Fanuc TP program (LS listing): test_parallel.ls

/PROG  test_parallel
/ATTR
COMMENT	= "18-08-08 11:10:22";
PROG_SIZE	= 0;
DEFAULT_GROUP	= 1, 1, *, *, *;
/APPL
    ARC Welding Equipment: 1, *, *, *, *;
/MN
   1:  CALL HOME_ALL;
   1:  UFRAME_NUM = 1;
   1:  UTOOL_NUM = 3;
   1:  COL GUARD ADJUST 150;
   1:  PR[91] = PR[90];
   1:  PR[GP1:91,1] = PR[GP1:90,1] + 65.993;
   1:  PR[GP1:91,2] = PR[GP1:90,2] + 95.281;
   1:  PR[GP1:91,3] = PR[GP1:90,3] + 0.900;
   1:L PR[91] 10mm/sec FINE;
   1:  PR[GP1:91,1] = PR[GP1:90,1] + 66.256;
   1:  PR[GP1:91,2] = PR[GP1:90,2] + 95.138;
   1:L PR[91] 10mm/sec FINE;
   1:  PR[GP1:91,1] = PR[GP1:90,1] + 70.899;
   1:  PR[GP1:91,2] = PR[GP1:90,2] + 93.080;
   1:L PR[91] 10mm/sec FINE;
   1:  PR[GP1:91,1] = PR[GP1:90,1] + 71.182;
   1:  PR[GP1:91,2] = PR[GP1:90,2] + 92.981;
   1:L PR[91] 10mm/sec FINE;
   1:  PR[GP1:91,1] = PR[GP1:90,1] + 71.477;
   1:  PR[GP1:91,2] = PR[GP1:90,2] + 92.931;
   1:L PR[91] 10mm/sec FINE;
   1:  PR[GP1:91,1] = PR[GP1:90,1] + 76.535;
   1:  PR[GP1:91,2] = PR[GP1:90,2] + 92.486;
   1:L PR[91] 10mm/sec FINE;
   1:  PR[GP1:91,1] = PR[GP1:90,1] + 76.835;
   1:  PR[GP1:91,2] = PR[GP1:90,2] + 92.484;
   1:L PR[91] 10mm/sec FINE;
   1:  PR[GP1:91,1] = PR[GP1:90,1] + 77.130;
   1:  PR[GP1:91,2] = PR[GP1:90,2] + 92.532;
   1:L PR[91] 10mm/sec FINE;
   1:  PR[GP1:91,1] = PR[GP1:90,1] + 82.061;
   1:  PR[GP1:91,2] = PR[GP1:90,2] + 93.748;
   1:L PR[91] 10mm/sec FINE;
   1:  PR[GP1:91,1] = PR[GP1:90,1] + 82.344;
   1:  PR[GP1:91,2] = PR[GP1:90,2] + 93.843;
   1:L PR[91] 10mm/sec FINE;
   1:  PR[GP1:91,1] = PR[GP1:90,1] + 82.609;
   1:  PR[GP1:91,2] = PR[GP1:90,2] + 93.984;
   1:L PR[91] 10mm/sec FINE;
   1:  PR[GP1:91,1] = PR[GP1:90,1] + 86.880;
   1:  PR[GP1:91,2] = PR[GP1:90,2] + 96.730;
   1:L PR[91] 10mm/sec FINE;
   1:  PR[GP1:91,1] = PR[GP1:90,1] + 87.118;
   1:  PR[GP1:91,2] = PR[GP1:90,2] + 96.912;
   1:L PR[91] 10mm/sec FINE;
   1:  PR[GP1:91,1] = PR[GP1:90,1] + 87.322;
   1:  PR[GP1:91,2] = PR[GP1:90,2] + 97.130;
   1:L PR[91] 10mm/sec FINE;
   1:  PR[GP1:91,1] = PR[GP1:90,1] + 90.476;
   1:  PR[GP1:91,2] = PR[GP1:90,2] + 101.111;
   1:L PR[91] 10mm/sec FINE;
   1:  PR[GP1:91,1] = PR[GP1:90,1] + 90.641;
   1:  PR[GP1:91,2] = PR[GP1:90,2] + 101.360;
   1:L PR[91] 10mm/sec FINE;
   1:  PR[GP1:91,1] = PR[GP1:90,1] + 90.764;
   1:  PR[GP1:91,2] = PR[GP1:90,2] + 101.633;
   1:L PR[91] 10mm/sec FINE;
   1:  PR[GP1:91,1] = PR[GP1:90,1] + 92.459;
   1:  PR[GP1:91,2] = PR[GP1:90,2] + 106.415;
   1:L PR[91] 10mm/sec FINE;
   1:  PR[GP1:91,1] = PR[GP1:90,1] + 92.544;
   1:  PR[GP1:91,2] = PR[GP1:90,2] + 106.735;
   1:L PR[91] 10mm/sec FINE;
   1:  PR[GP1:91,1] = PR[GP1:90,1] + 93.026;
   1:  PR[GP1:91,2] = PR[GP1:90,2] + 107.850;
   1:L PR[91] 10mm/sec FINE;
   1:  PR[GP1:91,1] = PR[GP1:90,1] + 93.981;
   1:  PR[GP1:91,2] = PR[GP1:90,2] + 108.650;
   1:L PR[91] 10mm/sec FINE;
   1:  PR[GP1:91,1] = PR[GP1:90,1] + 95.171;
   1:  PR[GP1:91,2] = PR[GP1:90,2] + 108.932;
   1:L PR[91] 10mm/sec FINE;
   1:  PR[GP1:91,1] = PR[GP1:90,1] + 95.835;
   1:L PR[91] 10mm/sec FINE;
   1:  PR[GP1:91,1] = PR[GP1:90,1] + 97.026;
   1:  PR[GP1:91,2] = PR[GP1:90,2] + 108.650;
   1:L PR[91] 10mm/sec FINE;
   1:  PR[GP1:91,1] = PR[GP1:90,1] + 97.981;
   1:  PR[GP1:91,2] = PR[GP1:90,2] + 107.850;
   1:L PR[91] 10mm/sec FINE;
   1:  PR[GP1:91,1] = PR[GP1:90,1] + 98.460;
   1:  PR[GP1:91,2] = PR[GP1:90,2] + 106.743;
   1:L PR[91] 10mm/sec FINE;
   1:  PR[GP1:91,1] = PR[GP1:90,1] + 100.166;
   1:  PR[GP1:91,2] = PR[GP1:90,2] + 101.928;
   1:L PR[91] 10mm/sec FINE;
   1:  PR[GP1:91,1] = PR[GP1:90,1] + 100.215;
   1:  PR[GP1:91,2] = PR[GP1:90,2] + 101.718;
   1:L PR[91] 10mm/sec FINE;
   1:  PR[GP1:91,1] = PR[GP1:90,1] + 100.280;
   1:  PR[GP1:91,2] = PR[GP1:90,2] + 101.535;
   1:L PR[91] 10mm/sec FINE;
   1:  PR[GP1:91,1] = PR[GP1:90,1] + 100.360;
   1:  PR[GP1:91,2] = PR[GP1:90,2] + 101.370;
   1:L PR[91] 10mm/sec FINE;
   1:  PR[GP1:91,1] = PR[GP1:90,1] + 103.517;
   1:  PR[GP1:91,2] = PR[GP1:90,2] + 97.385;
   1:L PR[91] 10mm/sec FINE;
   1:  PR[GP1:91,1] = PR[GP1:90,1] + 103.631;
   1:  PR[GP1:91,2] = PR[GP1:90,2] + 97.202;
   1:L PR[91] 10mm/sec FINE;
   1:  PR[GP1:91,1] = PR[GP1:90,1] + 103.752;
   1:  PR[GP1:91,2] = PR[GP1:90,2] + 97.049;
   1:L PR[91] 10mm/sec FINE;
   1:  PR[GP1:91,1] = PR[GP1:90,1] + 103.881;
   1:  PR[GP1:91,2] = PR[GP1:90,2] + 96.919;
   1:L PR[91] 10mm/sec FINE;
   1:  PR[GP1:91,1] = PR[GP1:90,1] + 108.157;
   1:  PR[GP1:91,2] = PR[GP1:90,2] + 94.170;
   1:L PR[91] 10mm/sec FINE;
   1:  PR[GP1:91,1] = PR[GP1:90,1] + 108.325;
   1:  PR[GP1:91,2] = PR[GP1:90,2] + 94.034;
   1:L PR[91] 10mm/sec FINE;
   1:  PR[GP1:91,1] = PR[GP1:90,1] + 108.488;
   1:  PR[GP1:91,2] = PR[GP1:90,2] + 93.929;
   1:L PR[91] 10mm/sec FINE;
   1:  PR[GP1:91,1] = PR[GP1:90,1] + 108.652;
   1:  PR[GP1:91,2] = PR[GP1:90,2] + 93.848;
   1:L PR[91] 10mm/sec FINE;
   1:  PR[GP1:91,1] = PR[GP1:90,1] + 113.587;
   1:  PR[GP1:91,2] = PR[GP1:90,2] + 92.631;
   1:L PR[91] 10mm/sec FINE;
   1:  PR[GP1:91,1] = PR[GP1:90,1] + 113.790;
   1:  PR[GP1:91,2] = PR[GP1:90,2] + 92.556;
   1:L PR[91] 10mm/sec FINE;
   1:  PR[GP1:91,1] = PR[GP1:90,1] + 113.978;
   1:  PR[GP1:91,2] = PR[GP1:90,2] + 92.510;
   1:L PR[91] 10mm/sec FINE;
   1:  PR[GP1:91,1] = PR[GP1:90,1] + 114.160;
   1:  PR[GP1:91,2] = PR[GP1:90,2] + 92.486;
   1:L PR[91] 10mm/sec FINE;
   1:  PR[GP1:91,1] = PR[GP1:90,1] + 119.224;
   1:  PR[GP1:91,2] = PR[GP1:90,2] + 92.931;
   1:L PR[91] 10mm/sec FINE;
   1:  PR[GP1:91,1] = PR[GP1:90,1] + 119.440;
   1:  PR[GP1:91,2] = PR[GP1:90,2] + 92.926;
   1:L PR[91] 10mm/sec FINE;
   1:  PR[GP1:91,1] = PR[GP1:90,1] + 119.633;
   1:  PR[GP1:91,2] = PR[GP1:90,2] + 92.943;
   1:L PR[91] 10mm/sec FINE;
   1:  PR[GP1:91,1] = PR[GP1:90,1] + 119.813;
   1:  PR[GP1:91,2] = PR[GP1:90,2] + 92.979;
   1:L PR[91] 10mm/sec FINE;
   1:  PR[GP1:91,1] = PR[GP1:90,1] + 124.460;
   1:  PR[GP1:91,2] = PR[GP1:90,2] + 95.038;
   1:L PR[91] 10mm/sec FINE;
   1:  PR[GP1:91,1] = PR[GP1:90,1] + 124.666;
   1:  PR[GP1:91,2] = PR[GP1:90,2] + 95.104;
   1:L PR[91] 10mm/sec FINE;
   1:  PR[GP1:91,1] = PR[GP1:90,1] + 124.844;
   1:  PR[GP1:91,2] = PR[GP1:90,2] + 95.182;
   1:L PR[91] 10mm/sec FINE;
   1:  PR[GP1:91,1] = PR[GP1:90,1] + 125.002;
   1:  PR[GP1:91,2] = PR[GP1:90,2] + 95.275;
   1:L PR[91] 10mm/sec FINE;
   1:  PR[GP1:91,1] = PR[GP1:90,1] + 128.734;
   1:  PR[GP1:91,2] = PR[GP1:90,2] + 98.728;
   1:L PR[91] 10mm/sec FINE;
   1:  PR[GP1:91,1] = PR[GP1:90,1] + 128.907;
   1:  PR[GP1:91,2] = PR[GP1:90,2] + 98.856;
   1:L PR[91] 10mm/sec FINE;
   1:  PR[GP1:91,1] = PR[GP1:90,1] + 129.050;
   1:  PR[GP1:91,2] = PR[GP1:90,2] + 98.988;
   1:L PR[91] 10mm/sec FINE;
   1:  PR[GP1:91,1] = PR[GP1:90,1] + 129.170;
   1:  PR[GP1:91,2] = PR[GP1:90,2] + 99.127;
   1:L PR[91] 10mm/sec FINE;
   1:  PR[GP1:91,1] = PR[GP1:90,1] + 131.584;
   1:  PR[GP1:91,2] = PR[GP1:90,2] + 103.603;
   1:L PR[91] 10mm/sec FINE;
   1:  PR[GP1:91,1] = PR[GP1:90,1] + 131.706;
   1:  PR[GP1:91,2] = PR[GP1:90,2] + 103.781;
   1:L PR[91] 10mm/sec FINE;
   1:  PR[GP1:91,1] = PR[GP1:90,1] + 131.798;
   1:  PR[GP1:91,2] = PR[GP1:90,2] + 103.951;
   1:L PR[91] 10mm/sec FINE;
   1:  PR[GP1:91,1] = PR[GP1:90,1] + 131.867;
   1:  PR[GP1:91,2] = PR[GP1:90,2] + 104.121;
   1:L PR[91] 10mm/sec FINE;
   1:  PR[GP1:91,1] = PR[GP1:90,1] + 132.702;
   1:  PR[GP1:91,2] = PR[GP1:90,2] + 109.139;
   1:L PR[91] 10mm/sec FINE;
   1:  PR[GP1:91,1] = PR[GP1:90,1] + 132.760;
   1:  PR[GP1:91,2] = PR[GP1:90,2] + 109.347;
   1:L PR[91] 10mm/sec FINE;
   1:  PR[GP1:91,1] = PR[GP1:90,1] + 132.792;
   1:  PR[GP1:91,2] = PR[GP1:90,2] + 109.538;
   1:L PR[91] 10mm/sec FINE;
   1:  PR[GP1:91,1] = PR[GP1:90,1] + 132.802;
   1:  PR[GP1:91,2] = PR[GP1:90,2] + 109.721;
   1:L PR[91] 10mm/sec FINE;
   1:  PR[GP1:91,1] = PR[GP1:90,1] + 131.968;
   1:  PR[GP1:91,2] = PR[GP1:90,2] + 114.734;
   1:L PR[91] 10mm/sec FINE;
   1:  PR[GP1:91,1] = PR[GP1:90,1] + 131.931;
   1:  PR[GP1:91,2] = PR[GP1:90,2] + 115.108;
   1:L PR[91] 10mm/sec FINE;
   1:  PR[GP1:91,1] = PR[GP1:90,1] + 131.829;
   1:  PR[GP1:91,2] = PR[GP1:90,2] + 115.442;
   1:L PR[91] 10mm/sec FINE;
   1:  PR[GP1:91,1] = PR[GP1:90,1] + 129.241;
   1:  PR[GP1:91,2] = PR[GP1:90,2] + 120.241;
   1:L PR[91] 10mm/sec FINE;
   1:  PR[GP1:91,1] = PR[GP1:90,1] + 129.179;
   1:  PR[GP1:91,2] = PR[GP1:90,2] + 120.327;
   1:L PR[91] 10mm/sec FINE;
   1:  PR[GP1:91,1] = PR[GP1:90,1] + 129.019;
   1:  PR[GP1:91,2] = PR[GP1:90,2] + 120.507;
   1:L PR[91] 10mm/sec FINE;
   1:  PR[GP1:91,1] = PR[GP1:90,1] + 125.292;
   1:  PR[GP1:91,2] = PR[GP1:90,2] + 123.956;
   1:L PR[91] 10mm/sec FINE;
   1:  PR[GP1:91,1] = PR[GP1:90,1] + 125.015;
   1:  PR[GP1:91,2] = PR[GP1:90,2] + 124.180;
   1:L PR[91] 10mm/sec FINE;
   1:  PR[GP1:91,1] = PR[GP1:90,1] + 120.376;
   1:  PR[GP1:91,2] = PR[GP1:90,2] + 126.236;
   1:L PR[91] 10mm/sec FINE;
   1:  PR[GP1:91,1] = PR[GP1:90,1] + 120.040;
   1:  PR[GP1:91,2] = PR[GP1:90,2] + 126.412;
   1:L PR[91] 10mm/sec FINE;
   1:  PR[GP1:91,1] = PR[GP1:90,1] + 119.820;
   1:  PR[GP1:91,2] = PR[GP1:90,2] + 126.484;
   1:L PR[91] 10mm/sec FINE;
   1:  PR[GP1:91,1] = PR[GP1:90,1] + 119.714;
   1:  PR[GP1:91,2] = PR[GP1:90,2] + 126.508;
   1:L PR[91] 10mm/sec FINE;
   1:  PR[GP1:91,1] = PR[GP1:90,1] + 114.278;
   1:  PR[GP1:91,2] = PR[GP1:90,2] + 126.985;
   1:L PR[91] 10mm/sec FINE;
   1:  PR[GP1:91,1] = PR[GP1:90,1] + 114.174;
   1:  PR[GP1:91,2] = PR[GP1:90,2] + 126.981;
   1:L PR[91] 10mm/sec FINE;
   1:  PR[GP1:91,1] = PR[GP1:90,1] + 113.934;
   1:  PR[GP1:91,2] = PR[GP1:90,2] + 126.946;
   1:L PR[91] 10mm/sec FINE;
   1:  PR[GP1:91,1] = PR[GP1:90,1] + 109.004;
   1:  PR[GP1:91,2] = PR[GP1:90,2] + 125.730;
   1:L PR[91] 10mm/sec FINE;
   1:  PR[GP1:91,1] = PR[GP1:90,1] + 108.669;
   1:  PR[GP1:91,2] = PR[GP1:90,2] + 125.623;
   1:L PR[91] 10mm/sec FINE;
   1:  PR[GP1:91,1] = PR[GP1:90,1] + 104.397;
   1:  PR[GP1:91,2] = PR[GP1:90,2] + 122.877;
   1:L PR[91] 10mm/sec FINE;
   1:  PR[GP1:91,1] = PR[GP1:90,1] + 104.066;
   1:  PR[GP1:91,2] = PR[GP1:90,2] + 122.693;
   1:L PR[91] 10mm/sec FINE;
   1:  PR[GP1:91,1] = PR[GP1:90,1] + 103.886;
   1:  PR[GP1:91,2] = PR[GP1:90,2] + 122.551;
   1:L PR[91] 10mm/sec FINE;
   1:  PR[GP1:91,1] = PR[GP1:90,1] + 103.806;
   1:  PR[GP1:91,2] = PR[GP1:90,2] + 122.474;
   1:L PR[91] 10mm/sec FINE;
   1:  PR[GP1:91,1] = PR[GP1:90,1] + 100.418;
   1:  PR[GP1:91,2] = PR[GP1:90,2] + 118.195;
   1:L PR[91] 10mm/sec FINE;
   1:  PR[GP1:91,1] = PR[GP1:90,1] + 100.366;
   1:  PR[GP1:91,2] = PR[GP1:90,2] + 118.108;
   1:L PR[91] 10mm/sec FINE;
   1:  PR[GP1:91,1] = PR[GP1:90,1] + 100.262;
   1:  PR[GP1:91,2] = PR[GP1:90,2] + 117.886;
   1:L PR[91] 10mm/sec FINE;
   1:  PR[GP1:91,1] = PR[GP1:90,1] + 98.568;
   1:  PR[GP1:91,2] = PR[GP1:90,2] + 113.104;
   1:L PR[91] 10mm/sec FINE;
   1:  PR[GP1:91,1] = PR[GP1:90,1] + 98.462;
   1:  PR[GP1:91,2] = PR[GP1:90,2] + 112.728;
   1:L PR[91] 10mm/sec FINE;
   1:  PR[GP1:91,1] = PR[GP1:90,1] + 97.981;
   1:  PR[GP1:91,2] = PR[GP1:90,2] + 111.615;
   1:L PR[91] 10mm/sec FINE;
   1:  PR[GP1:91,1] = PR[GP1:90,1] + 97.026;
   1:  PR[GP1:91,2] = PR[GP1:90,2] + 110.814;
   1:L PR[91] 10mm/sec FINE;
   1:  PR[GP1:91,1] = PR[GP1:90,1] + 95.835;
   1:  PR[GP1:91,2] = PR[GP1:90,2] + 110.532;
   1:L PR[91] 10mm/sec FINE;
   1:  PR[GP1:91,1] = PR[GP1:90,1] + 95.171;
   1:L PR[91] 10mm/sec FINE;
   1:  PR[GP1:91,1] = PR[GP1:90,1] + 93.981;
   1:  PR[GP1:91,2] = PR[GP1:90,2] + 110.814;
   1:L PR[91] 10mm/sec FINE;
   1:  PR[GP1:91,1] = PR[GP1:90,1] + 93.026;
   1:  PR[GP1:91,2] = PR[GP1:90,2] + 111.615;
   1:L PR[91] 10mm/sec FINE;
   1:  PR[GP1:91,1] = PR[GP1:90,1] + 92.547;
   1:  PR[GP1:91,2] = PR[GP1:90,2] + 112.721;
   1:L PR[91] 10mm/sec FINE;
   1:  PR[GP1:91,1] = PR[GP1:90,1] + 90.842;
   1:  PR[GP1:91,2] = PR[GP1:90,2] + 117.534;
   1:L PR[91] 10mm/sec FINE;
   1:  PR[GP1:91,1] = PR[GP1:90,1] + 90.761;
   1:  PR[GP1:91,2] = PR[GP1:90,2] + 117.840;
   1:L PR[91] 10mm/sec FINE;
   1:  PR[GP1:91,1] = PR[GP1:90,1] + 90.645;
   1:  PR[GP1:91,2] = PR[GP1:90,2] + 118.097;
   1:L PR[91] 10mm/sec FINE;
   1:  PR[GP1:91,1] = PR[GP1:90,1] + 87.492;
   1:  PR[GP1:91,2] = PR[GP1:90,2] + 122.078;
   1:L PR[91] 10mm/sec FINE;
   1:  PR[GP1:91,1] = PR[GP1:90,1] + 87.317;
   1:  PR[GP1:91,2] = PR[GP1:90,2] + 122.340;
   1:L PR[91] 10mm/sec FINE;
   1:  PR[GP1:91,1] = PR[GP1:90,1] + 87.123;
   1:  PR[GP1:91,2] = PR[GP1:90,2] + 122.547;
   1:L PR[91] 10mm/sec FINE;
   1:  PR[GP1:91,1] = PR[GP1:90,1] + 82.852;
   1:  PR[GP1:91,2] = PR[GP1:90,2] + 125.293;
   1:L PR[91] 10mm/sec FINE;
   1:  PR[GP1:91,1] = PR[GP1:90,1] + 82.601;
   1:  PR[GP1:91,2] = PR[GP1:90,2] + 125.485;
   1:L PR[91] 10mm/sec FINE;
   1:  PR[GP1:91,1] = PR[GP1:90,1] + 82.352;
   1:  PR[GP1:91,2] = PR[GP1:90,2] + 125.617;
   1:L PR[91] 10mm/sec FINE;
   1:  PR[GP1:91,1] = PR[GP1:90,1] + 77.421;
   1:  PR[GP1:91,2] = PR[GP1:90,2] + 126.834;
   1:L PR[91] 10mm/sec FINE;
   1:  PR[GP1:91,1] = PR[GP1:90,1] + 77.122;
   1:  PR[GP1:91,2] = PR[GP1:90,2] + 126.934;
   1:L PR[91] 10mm/sec FINE;
   1:  PR[GP1:91,1] = PR[GP1:90,1] + 76.843;
   1:  PR[GP1:91,2] = PR[GP1:90,2] + 126.979;
   1:L PR[91] 10mm/sec FINE;
   1:  PR[GP1:91,1] = PR[GP1:90,1] + 71.784;
   1:  PR[GP1:91,2] = PR[GP1:90,2] + 126.534;
   1:L PR[91] 10mm/sec FINE;
   1:  PR[GP1:91,1] = PR[GP1:90,1] + 71.468;
   1:  PR[GP1:91,2] = PR[GP1:90,2] + 126.532;
   1:L PR[91] 10mm/sec FINE;
   1:  PR[GP1:91,1] = PR[GP1:90,1] + 71.190;
   1:  PR[GP1:91,2] = PR[GP1:90,2] + 126.484;
   1:L PR[91] 10mm/sec FINE;
   1:  PR[GP1:91,1] = PR[GP1:90,1] + 66.547;
   1:  PR[GP1:91,2] = PR[GP1:90,2] + 124.426;
   1:L PR[91] 10mm/sec FINE;
   1:  PR[GP1:91,1] = PR[GP1:90,1] + 66.249;
   1:  PR[GP1:91,2] = PR[GP1:90,2] + 124.323;
   1:L PR[91] 10mm/sec FINE;
   1:  PR[GP1:91,1] = PR[GP1:90,1] + 66.001;
   1:  PR[GP1:91,2] = PR[GP1:90,2] + 124.187;
   1:L PR[91] 10mm/sec FINE;
   1:  PR[GP1:91,1] = PR[GP1:90,1] + 62.274;
   1:  PR[GP1:91,2] = PR[GP1:90,2] + 120.737;
   1:L PR[91] 10mm/sec FINE;
   1:  PR[GP1:91,1] = PR[GP1:90,1] + 62.025;
   1:  PR[GP1:91,2] = PR[GP1:90,2] + 120.542;
   1:L PR[91] 10mm/sec FINE;
   1:  PR[GP1:91,1] = PR[GP1:90,1] + 61.834;
   1:  PR[GP1:91,2] = PR[GP1:90,2] + 120.334;
   1:L PR[91] 10mm/sec FINE;
   1:  PR[GP1:91,1] = PR[GP1:90,1] + 59.424;
   1:  PR[GP1:91,2] = PR[GP1:90,2] + 115.863;
   1:L PR[91] 10mm/sec FINE;
   1:  PR[GP1:91,1] = PR[GP1:90,1] + 59.252;
   1:  PR[GP1:91,2] = PR[GP1:90,2] + 115.598;
   1:L PR[91] 10mm/sec FINE;
   1:  PR[GP1:91,1] = PR[GP1:90,1] + 59.139;
   1:  PR[GP1:91,2] = PR[GP1:90,2] + 115.339;
   1:L PR[91] 10mm/sec FINE;
   1:  PR[GP1:91,1] = PR[GP1:90,1] + 58.305;
   1:  PR[GP1:91,2] = PR[GP1:90,2] + 110.328;
   1:L PR[91] 10mm/sec FINE;
   1:  PR[GP1:91,1] = PR[GP1:90,1] + 58.228;
   1:  PR[GP1:91,2] = PR[GP1:90,2] + 110.022;
   1:L PR[91] 10mm/sec FINE;
   1:  PR[GP1:91,1] = PR[GP1:90,1] + 58.205;
   1:  PR[GP1:91,2] = PR[GP1:90,2] + 109.741;
   1:L PR[91] 10mm/sec FINE;
   1:  PR[GP1:91,1] = PR[GP1:90,1] + 59.038;
   1:  PR[GP1:91,2] = PR[GP1:90,2] + 104.730;
   1:L PR[91] 10mm/sec FINE;
   1:  PR[GP1:91,1] = PR[GP1:90,1] + 59.064;
   1:  PR[GP1:91,2] = PR[GP1:90,2] + 104.415;
   1:L PR[91] 10mm/sec FINE;
   1:  PR[GP1:91,1] = PR[GP1:90,1] + 59.135;
   1:  PR[GP1:91,2] = PR[GP1:90,2] + 104.133;
   1:L PR[91] 10mm/sec FINE;
   1:  PR[GP1:91,1] = PR[GP1:90,1] + 59.255;
   1:  PR[GP1:91,2] = PR[GP1:90,2] + 103.859;
   1:L PR[91] 10mm/sec FINE;
   1:  PR[GP1:91,1] = PR[GP1:90,1] + 61.665;
   1:  PR[GP1:91,2] = PR[GP1:90,2] + 99.388;
   1:L PR[91] 10mm/sec FINE;
   1:  PR[GP1:91,1] = PR[GP1:90,1] + 61.829;
   1:  PR[GP1:91,2] = PR[GP1:90,2] + 99.137;
   1:L PR[91] 10mm/sec FINE;
   1:  PR[GP1:91,1] = PR[GP1:90,1] + 62.031;
   1:  PR[GP1:91,2] = PR[GP1:90,2] + 98.916;
   1:L PR[91] 10mm/sec FINE;
   1:  PR[GP1:91,1] = PR[GP1:90,1] + 65.758;
   1:  PR[GP1:91,2] = PR[GP1:90,2] + 95.466;
   1:L PR[91] 10mm/sec FINE;
   1:  PR[GP1:91,1] = PR[GP1:90,1] + 65.993;
   1:  PR[GP1:91,2] = PR[GP1:90,2] + 95.281;
   1:L PR[91] 10mm/sec FINE;
   1:  PR[GP1:91,1] = PR[GP1:90,1] + 66.856;
   1:  PR[GP1:91,2] = PR[GP1:90,2] + 94.811;
   1:  PR[GP1:91,3] = PR[GP1:90,3] + 1.900;
   1:L PR[91] 10mm/sec FINE;
   1:  PR[GP1:91,1] = PR[GP1:90,1] + 70.252;
   1:  PR[GP1:91,2] = PR[GP1:90,2] + 93.305;
   1:L PR[91] 10mm/sec FINE;
   1:  PR[GP1:91,1] = PR[GP1:90,1] + 71.181;
   1:  PR[GP1:91,2] = PR[GP1:90,2] + 92.982;
   1:L PR[91] 10mm/sec FINE;
   1:  PR[GP1:91,1] = PR[GP1:90,1] + 72.150;
   1:  PR[GP1:91,2] = PR[GP1:90,2] + 92.815;
   1:L PR[91] 10mm/sec FINE;
   1:  PR[GP1:91,1] = PR[GP1:90,1] + 75.850;
   1:  PR[GP1:91,2] = PR[GP1:90,2] + 92.490;
   1:L PR[91] 10mm/sec FINE;
   1:  PR[GP1:91,1] = PR[GP1:90,1] + 76.834;
   1:  PR[GP1:91,2] = PR[GP1:90,2] + 92.484;
   1:L PR[91] 10mm/sec FINE;
   1:  PR[GP1:91,1] = PR[GP1:90,1] + 77.804;
   1:  PR[GP1:91,2] = PR[GP1:90,2] + 92.640;
   1:L PR[91] 10mm/sec FINE;
   1:  PR[GP1:91,1] = PR[GP1:90,1] + 81.411;
   1:  PR[GP1:91,2] = PR[GP1:90,2] + 93.530;
   1:L PR[91] 10mm/sec FINE;
   1:  PR[GP1:91,1] = PR[GP1:90,1] + 82.343;
   1:  PR[GP1:91,2] = PR[GP1:90,2] + 93.843;
   1:L PR[91] 10mm/sec FINE;
   1:  PR[GP1:91,1] = PR[GP1:90,1] + 83.212;
   1:  PR[GP1:91,2] = PR[GP1:90,2] + 94.304;
   1:L PR[91] 10mm/sec FINE;
   1:  PR[GP1:91,1] = PR[GP1:90,1] + 86.336;
   1:  PR[GP1:91,2] = PR[GP1:90,2] + 96.313;
   1:L PR[91] 10mm/sec FINE;
   1:  PR[GP1:91,1] = PR[GP1:90,1] + 87.117;
   1:  PR[GP1:91,2] = PR[GP1:90,2] + 96.911;
   1:L PR[91] 10mm/sec FINE;
   1:  PR[GP1:91,1] = PR[GP1:90,1] + 87.789;
   1:  PR[GP1:91,2] = PR[GP1:90,2] + 97.629;
   1:L PR[91] 10mm/sec FINE;
   1:  PR[GP1:91,1] = PR[GP1:90,1] + 90.096;
   1:  PR[GP1:91,2] = PR[GP1:90,2] + 100.540;
   1:L PR[91] 10mm/sec FINE;
   1:  PR[GP1:91,1] = PR[GP1:90,1] + 90.641;
   1:  PR[GP1:91,2] = PR[GP1:90,2] + 101.359;
   1:L PR[91] 10mm/sec FINE;
   1:  PR[GP1:91,1] = PR[GP1:90,1] + 91.045;
   1:  PR[GP1:91,2] = PR[GP1:90,2] + 102.255;
   1:L PR[91] 10mm/sec FINE;
   1:  PR[GP1:91,1] = PR[GP1:90,1] + 92.284;
   1:  PR[GP1:91,2] = PR[GP1:90,2] + 105.754;
   1:L PR[91] 10mm/sec FINE;
   1:  PR[GP1:91,1] = PR[GP1:90,1] + 92.544;
   1:  PR[GP1:91,2] = PR[GP1:90,2] + 106.735;
   1:L PR[91] 10mm/sec FINE;
   1:  PR[GP1:91,1] = PR[GP1:90,1] + 93.026;
   1:  PR[GP1:91,2] = PR[GP1:90,2] + 107.850;
   1:L PR[91] 10mm/sec FINE;
   1:  PR[GP1:91,1] = PR[GP1:90,1] + 93.981;
   1:  PR[GP1:91,2] = PR[GP1:90,2] + 108.650;
   1:L PR[91] 10mm/sec FINE;
   1:  PR[GP1:91,1] = PR[GP1:90,1] + 95.171;
   1:  PR[GP1:91,2] = PR[GP1:90,2] + 108.932;
   1:L PR[91] 10mm/sec FINE;
   1:  PR[GP1:91,1] = PR[GP1:90,1] + 95.835;
   1:L PR[91] 10mm/sec FINE;
   1:  PR[GP1:91,1] = PR[GP1:90,1] + 97.025;
   1:  PR[GP1:91,2] = PR[GP1:90,2] + 108.650;
   1:L PR[91] 10mm/sec FINE;
   1:  PR[GP1:91,1] = PR[GP1:90,1] + 97.981;
   1:  PR[GP1:91,2] = PR[GP1:90,2] + 107.850;
   1:L PR[91] 10mm/sec FINE;
   1:  PR[GP1:91,1] = PR[GP1:90,1] + 98.460;
   1:  PR[GP1:91,2] = PR[GP1:90,2] + 106.743;
   1:L PR[91] 10mm/sec FINE;
   1:  PR[GP1:91,1] = PR[GP1:90,1] + 99.711;
   1:  PR[GP1:91,2] = PR[GP1:90,2] + 103.212;
   1:L PR[91] 10mm/sec FINE;
   1:  PR[GP1:91,1] = PR[GP1:90,1] + 99.865;
   1:  PR[GP1:91,2] = PR[GP1:90,2] + 102.558;
   1:L PR[91] 10mm/sec FINE;
   1:  PR[GP1:91,1] = PR[GP1:90,1] + 100.082;
   1:  PR[GP1:91,2] = PR[GP1:90,2] + 101.944;
   1:L PR[91] 10mm/sec FINE;
   1:  PR[GP1:91,1] = PR[GP1:90,1] + 100.360;
   1:  PR[GP1:91,2] = PR[GP1:90,2] + 101.369;
   1:L PR[91] 10mm/sec FINE;
   1:  PR[GP1:91,1] = PR[GP1:90,1] + 102.670;
   1:  PR[GP1:91,2] = PR[GP1:90,2] + 98.452;
   1:L PR[91] 10mm/sec FINE;
   1:  PR[GP1:91,1] = PR[GP1:90,1] + 103.028;
   1:  PR[GP1:91,2] = PR[GP1:90,2] + 97.883;
   1:L PR[91] 10mm/sec FINE;
   1:  PR[GP1:91,1] = PR[GP1:90,1] + 103.432;
   1:  PR[GP1:91,2] = PR[GP1:90,2] + 97.373;
   1:L PR[91] 10mm/sec FINE;
   1:  PR[GP1:91,1] = PR[GP1:90,1] + 103.882;
   1:  PR[GP1:91,2] = PR[GP1:90,2] + 96.919;
   1:L PR[91] 10mm/sec FINE;
   1:  PR[GP1:91,1] = PR[GP1:90,1] + 107.011;
   1:  PR[GP1:91,2] = PR[GP1:90,2] + 94.907;
   1:L PR[91] 10mm/sec FINE;
   1:  PR[GP1:91,1] = PR[GP1:90,1] + 107.533;
   1:  PR[GP1:91,2] = PR[GP1:90,2] + 94.484;
   1:L PR[91] 10mm/sec FINE;
   1:  PR[GP1:91,1] = PR[GP1:90,1] + 108.080;
   1:  PR[GP1:91,2] = PR[GP1:90,2] + 94.132;
   1:L PR[91] 10mm/sec FINE;
   1:  PR[GP1:91,1] = PR[GP1:90,1] + 108.653;
   1:  PR[GP1:91,2] = PR[GP1:90,2] + 93.847;
   1:L PR[91] 10mm/sec FINE;
   1:  PR[GP1:91,1] = PR[GP1:90,1] + 112.265;
   1:  PR[GP1:91,2] = PR[GP1:90,2] + 92.957;
   1:L PR[91] 10mm/sec FINE;
   1:  PR[GP1:91,1] = PR[GP1:90,1] + 112.896;
   1:  PR[GP1:91,2] = PR[GP1:90,2] + 92.725;
   1:L PR[91] 10mm/sec FINE;
   1:  PR[GP1:91,1] = PR[GP1:90,1] + 113.527;
   1:  PR[GP1:91,2] = PR[GP1:90,2] + 92.570;
   1:L PR[91] 10mm/sec FINE;
   1:  PR[GP1:91,1] = PR[GP1:90,1] + 114.161;
   1:  PR[GP1:91,2] = PR[GP1:90,2] + 92.486;
   1:L PR[91] 10mm/sec FINE;
   1:  PR[GP1:91,1] = PR[GP1:90,1] + 117.867;
   1:  PR[GP1:91,2] = PR[GP1:90,2] + 92.811;
   1:L PR[91] 10mm/sec FINE;
   1:  PR[GP1:91,1] = PR[GP1:90,1] + 118.539;
   1:  PR[GP1:91,2] = PR[GP1:90,2] + 92.796;
   1:L PR[91] 10mm/sec FINE;
   1:  PR[GP1:91,1] = PR[GP1:90,1] + 119.187;
   1:  PR[GP1:91,2] = PR[GP1:90,2] + 92.853;
   1:L PR[91] 10mm/sec FINE;
   1:  PR[GP1:91,1] = PR[GP1:90,1] + 119.814;
   1:  PR[GP1:91,2] = PR[GP1:90,2] + 92.979;
   1:L PR[91] 10mm/sec FINE;
   1:  PR[GP1:91,1] = PR[GP1:90,1] + 123.215;
   1:  PR[GP1:91,2] = PR[GP1:90,2] + 94.486;
   1:L PR[91] 10mm/sec FINE;
   1:  PR[GP1:91,1] = PR[GP1:90,1] + 123.856;
   1:  PR[GP1:91,2] = PR[GP1:90,2] + 94.690;
   1:L PR[91] 10mm/sec FINE;
   1:  PR[GP1:91,1] = PR[GP1:90,1] + 124.451;
   1:  PR[GP1:91,2] = PR[GP1:90,2] + 94.954;
   1:L PR[91] 10mm/sec FINE;
   1:  PR[GP1:91,1] = PR[GP1:90,1] + 125.003;
   1:  PR[GP1:91,2] = PR[GP1:90,2] + 95.275;
   1:L PR[91] 10mm/sec FINE;
   1:  PR[GP1:91,1] = PR[GP1:90,1] + 127.734;
   1:  PR[GP1:91,2] = PR[GP1:90,2] + 97.802;
   1:L PR[91] 10mm/sec FINE;
   1:  PR[GP1:91,1] = PR[GP1:90,1] + 128.275;
   1:  PR[GP1:91,2] = PR[GP1:90,2] + 98.202;
   1:L PR[91] 10mm/sec FINE;
   1:  PR[GP1:91,1] = PR[GP1:90,1] + 128.752;
   1:  PR[GP1:91,2] = PR[GP1:90,2] + 98.644;
   1:L PR[91] 10mm/sec FINE;
   1:  PR[GP1:91,1] = PR[GP1:90,1] + 129.171;
   1:  PR[GP1:91,2] = PR[GP1:90,2] + 99.128;
   1:L PR[91] 10mm/sec FINE;
   1:  PR[GP1:91,1] = PR[GP1:90,1] + 130.937;
   1:  PR[GP1:91,2] = PR[GP1:90,2] + 102.403;
   1:L PR[91] 10mm/sec FINE;
   1:  PR[GP1:91,1] = PR[GP1:90,1] + 131.319;
   1:  PR[GP1:91,2] = PR[GP1:90,2] + 102.957;
   1:L PR[91] 10mm/sec FINE;
   1:  PR[GP1:91,1] = PR[GP1:90,1] + 131.628;
   1:  PR[GP1:91,2] = PR[GP1:90,2] + 103.529;
   1:L PR[91] 10mm/sec FINE;
   1:  PR[GP1:91,1] = PR[GP1:90,1] + 131.867;
   1:  PR[GP1:91,2] = PR[GP1:90,2] + 104.122;
   1:L PR[91] 10mm/sec FINE;
   1:  PR[GP1:91,1] = PR[GP1:90,1] + 132.478;
   1:  PR[GP1:91,2] = PR[GP1:90,2] + 107.794;
   1:L PR[91] 10mm/sec FINE;
   1:  PR[GP1:91,1] = PR[GP1:90,1] + 132.661;
   1:  PR[GP1:91,2] = PR[GP1:90,2] + 108.441;
   1:L PR[91] 10mm/sec FINE;
   1:  PR[GP1:91,1] = PR[GP1:90,1] + 132.767;
   1:  PR[GP1:91,2] = PR[GP1:90,2] + 109.083;
   1:L PR[91] 10mm/sec FINE;
   1:  PR[GP1:91,1] = PR[GP1:90,1] + 132.802;
   1:  PR[GP1:91,2] = PR[GP1:90,2] + 109.721;
   1:L PR[91] 10mm/sec FINE;
   1:  PR[GP1:91,1] = PR[GP1:90,1] + 132.192;
   1:  PR[GP1:91,2] = PR[GP1:90,2] + 113.389;
   1:L PR[91] 10mm/sec FINE;
   1:  PR[GP1:91,1] = PR[GP1:90,1] + 132.074;
   1:  PR[GP1:91,2] = PR[GP1:90,2] + 114.582;
   1:L PR[91] 10mm/sec FINE;
   1:  PR[GP1:91,1] = PR[GP1:90,1] + 131.870;
   1:  PR[GP1:91,2] = PR[GP1:90,2] + 115.335;
   1:L PR[91] 10mm/sec FINE;
   1:  PR[GP1:91,1] = PR[GP1:90,1] + 131.735;
   1:  PR[GP1:91,2] = PR[GP1:90,2] + 115.692;
   1:L PR[91] 10mm/sec FINE;
   1:  PR[GP1:91,1] = PR[GP1:90,1] + 129.402;
   1:  PR[GP1:91,2] = PR[GP1:90,2] + 120.020;
   1:L PR[91] 10mm/sec FINE;
   1:  PR[GP1:91,1] = PR[GP1:90,1] + 129.180;
   1:  PR[GP1:91,2] = PR[GP1:90,2] + 120.326;
   1:L PR[91] 10mm/sec FINE;
   1:  PR[GP1:91,1] = PR[GP1:90,1] + 128.656;
   1:  PR[GP1:91,2] = PR[GP1:90,2] + 120.918;
   1:L PR[91] 10mm/sec FINE;
   1:  PR[GP1:91,1] = PR[GP1:90,1] + 125.929;
   1:  PR[GP1:91,2] = PR[GP1:90,2] + 123.441;
   1:L PR[91] 10mm/sec FINE;
   1:  PR[GP1:91,1] = PR[GP1:90,1] + 125.014;
   1:  PR[GP1:91,2] = PR[GP1:90,2] + 124.181;
   1:L PR[91] 10mm/sec FINE;
   1:  PR[GP1:91,1] = PR[GP1:90,1] + 121.621;
   1:  PR[GP1:91,2] = PR[GP1:90,2] + 125.685;
   1:L PR[91] 10mm/sec FINE;
   1:  PR[GP1:91,1] = PR[GP1:90,1] + 120.557;
   1:  PR[GP1:91,2] = PR[GP1:90,2] + 126.242;
   1:L PR[91] 10mm/sec FINE;
   1:  PR[GP1:91,1] = PR[GP1:90,1] + 119.822;
   1:  PR[GP1:91,2] = PR[GP1:90,2] + 126.484;
   1:L PR[91] 10mm/sec FINE;
   1:  PR[GP1:91,1] = PR[GP1:90,1] + 119.443;
   1:  PR[GP1:91,2] = PR[GP1:90,2] + 126.568;
   1:L PR[91] 10mm/sec FINE;
   1:  PR[GP1:91,1] = PR[GP1:90,1] + 114.547;
   1:  PR[GP1:91,2] = PR[GP1:90,2] + 126.997;
   1:L PR[91] 10mm/sec FINE;
   1:  PR[GP1:91,1] = PR[GP1:90,1] + 114.176;
   1:  PR[GP1:91,2] = PR[GP1:90,2] + 126.981;
   1:L PR[91] 10mm/sec FINE;
   1:  PR[GP1:91,1] = PR[GP1:90,1] + 113.387;
   1:  PR[GP1:91,2] = PR[GP1:90,2] + 126.867;
   1:L PR[91] 10mm/sec FINE;
   1:  PR[GP1:91,1] = PR[GP1:90,1] + 109.781;
   1:  PR[GP1:91,2] = PR[GP1:90,2] + 125.977;
   1:L PR[91] 10mm/sec FINE;
   1:  PR[GP1:91,1] = PR[GP1:90,1] + 108.670;
   1:  PR[GP1:91,2] = PR[GP1:90,2] + 125.623;
   1:L PR[91] 10mm/sec FINE;
   1:  PR[GP1:91,1] = PR[GP1:90,1] + 105.538;
   1:  PR[GP1:91,2] = PR[GP1:90,2] + 123.612;
   1:L PR[91] 10mm/sec FINE;
   1:  PR[GP1:91,1] = PR[GP1:90,1] + 104.489;
   1:  PR[GP1:91,2] = PR[GP1:90,2] + 123.029;
   1:L PR[91] 10mm/sec FINE;
   1:  PR[GP1:91,1] = PR[GP1:90,1] + 103.887;
   1:  PR[GP1:91,2] = PR[GP1:90,2] + 122.552;
   1:L PR[91] 10mm/sec FINE;
   1:  PR[GP1:91,1] = PR[GP1:90,1] + 103.604;
   1:  PR[GP1:91,2] = PR[GP1:90,2] + 122.278;
   1:L PR[91] 10mm/sec FINE;
   1:  PR[GP1:91,1] = PR[GP1:90,1] + 100.554;
   1:  PR[GP1:91,2] = PR[GP1:90,2] + 118.423;
   1:L PR[91] 10mm/sec FINE;
   1:  PR[GP1:91,1] = PR[GP1:90,1] + 100.367;
   1:  PR[GP1:91,2] = PR[GP1:90,2] + 118.109;
   1:L PR[91] 10mm/sec FINE;
   1:  PR[GP1:91,1] = PR[GP1:90,1] + 100.026;
   1:  PR[GP1:91,2] = PR[GP1:90,2] + 117.382;
   1:L PR[91] 10mm/sec FINE;
   1:  PR[GP1:91,1] = PR[GP1:90,1] + 98.786;
   1:  PR[GP1:91,2] = PR[GP1:90,2] + 113.883;
   1:L PR[91] 10mm/sec FINE;
   1:  PR[GP1:91,1] = PR[GP1:90,1] + 98.462;
   1:  PR[GP1:91,2] = PR[GP1:90,2] + 112.728;
   1:L PR[91] 10mm/sec FINE;
   1:  PR[GP1:91,1] = PR[GP1:90,1] + 97.981;
   1:  PR[GP1:91,2] = PR[GP1:90,2] + 111.615;
   1:L PR[91] 10mm/sec FINE;
   1:  PR[GP1:91,1] = PR[GP1:90,1] + 97.025;
   1:  PR[GP1:91,2] = PR[GP1:90,2] + 110.814;
   1:L PR[91] 10mm/sec FINE;
   1:  PR[GP1:91,1] = PR[GP1:90,1] + 95.835;
   1:  PR[GP1:91,2] = PR[GP1:90,2] + 110.532;
   1:L PR[91] 10mm/sec FINE;
   1:  PR[GP1:91,1] = PR[GP1:90,1] + 95.171;
   1:L PR[91] 10mm/sec FINE;
   1:  PR[GP1:91,1] = PR[GP1:90,1] + 93.981;
   1:  PR[GP1:91,2] = PR[GP1:90,2] + 110.814;
   1:L PR[91] 10mm/sec FINE;
   1:  PR[GP1:91,1] = PR[GP1:90,1] + 93.026;
   1:  PR[GP1:91,2] = PR[GP1:90,2] + 111.615;
   1:L PR[91] 10mm/sec FINE;
   1:  PR[GP1:91,1] = PR[GP1:90,1] + 92.547;
   1:  PR[GP1:91,2] = PR[GP1:90,2] + 112.721;
   1:L PR[91] 10mm/sec FINE;
   1:  PR[GP1:91,1] = PR[GP1:90,1] + 91.297;
   1:  PR[GP1:91,2] = PR[GP1:90,2] + 116.250;
   1:L PR[91] 10mm/sec FINE;
   1:  PR[GP1:91,1] = PR[GP1:90,1] + 91.041;
   1:  PR[GP1:91,2] = PR[GP1:90,2] + 117.217;
   1:L PR[91] 10mm/sec FINE;
   1:  PR[GP1:91,1] = PR[GP1:90,1] + 90.644;
   1:  PR[GP1:91,2] = PR[GP1:90,2] + 118.098;
   1:L PR[91] 10mm/sec FINE;
   1:  PR[GP1:91,1] = PR[GP1:90,1] + 88.338;
   1:  PR[GP1:91,2] = PR[GP1:90,2] + 121.010;
   1:L PR[91] 10mm/sec FINE;
   1:  PR[GP1:91,1] = PR[GP1:90,1] + 87.783;
   1:  PR[GP1:91,2] = PR[GP1:90,2] + 121.842;
   1:L PR[91] 10mm/sec FINE;
   1:  PR[GP1:91,1] = PR[GP1:90,1] + 87.123;
   1:  PR[GP1:91,2] = PR[GP1:90,2] + 122.548;
   1:L PR[91] 10mm/sec FINE;
   1:  PR[GP1:91,1] = PR[GP1:90,1] + 83.998;
   1:  PR[GP1:91,2] = PR[GP1:90,2] + 124.556;
   1:L PR[91] 10mm/sec FINE;
   1:  PR[GP1:91,1] = PR[GP1:90,1] + 83.204;
   1:  PR[GP1:91,2] = PR[GP1:90,2] + 125.164;
   1:L PR[91] 10mm/sec FINE;
   1:  PR[GP1:91,1] = PR[GP1:90,1] + 82.351;
   1:  PR[GP1:91,2] = PR[GP1:90,2] + 125.618;
   1:L PR[91] 10mm/sec FINE;
   1:  PR[GP1:91,1] = PR[GP1:90,1] + 78.744;
   1:  PR[GP1:91,2] = PR[GP1:90,2] + 126.508;
   1:L PR[91] 10mm/sec FINE;
   1:  PR[GP1:91,1] = PR[GP1:90,1] + 77.796;
   1:  PR[GP1:91,2] = PR[GP1:90,2] + 126.826;
   1:L PR[91] 10mm/sec FINE;
   1:  PR[GP1:91,1] = PR[GP1:90,1] + 76.842;
   1:  PR[GP1:91,2] = PR[GP1:90,2] + 126.979;
   1:L PR[91] 10mm/sec FINE;
   1:  PR[GP1:91,1] = PR[GP1:90,1] + 73.141;
   1:  PR[GP1:91,2] = PR[GP1:90,2] + 126.654;
   1:L PR[91] 10mm/sec FINE;
   1:  PR[GP1:91,1] = PR[GP1:90,1] + 72.142;
   1:  PR[GP1:91,2] = PR[GP1:90,2] + 126.648;
   1:L PR[91] 10mm/sec FINE;
   1:  PR[GP1:91,1] = PR[GP1:90,1] + 71.189;
   1:  PR[GP1:91,2] = PR[GP1:90,2] + 126.484;
   1:L PR[91] 10mm/sec FINE;
   1:  PR[GP1:91,1] = PR[GP1:90,1] + 67.793;
   1:  PR[GP1:91,2] = PR[GP1:90,2] + 124.979;
   1:L PR[91] 10mm/sec FINE;
   1:  PR[GP1:91,1] = PR[GP1:90,1] + 66.848;
   1:  PR[GP1:91,2] = PR[GP1:90,2] + 124.650;
   1:L PR[91] 10mm/sec FINE;
   1:  PR[GP1:91,1] = PR[GP1:90,1] + 66.000;
   1:  PR[GP1:91,2] = PR[GP1:90,2] + 124.187;
   1:L PR[91] 10mm/sec FINE;
   1:  PR[GP1:91,1] = PR[GP1:90,1] + 63.273;
   1:  PR[GP1:91,2] = PR[GP1:90,2] + 121.663;
   1:L PR[91] 10mm/sec FINE;
   1:  PR[GP1:91,1] = PR[GP1:90,1] + 62.487;
   1:  PR[GP1:91,2] = PR[GP1:90,2] + 121.046;
   1:L PR[91] 10mm/sec FINE;
   1:  PR[GP1:91,1] = PR[GP1:90,1] + 61.834;
   1:  PR[GP1:91,2] = PR[GP1:90,2] + 120.333;
   1:L PR[91] 10mm/sec FINE;
   1:  PR[GP1:91,1] = PR[GP1:90,1] + 60.071;
   1:  PR[GP1:91,2] = PR[GP1:90,2] + 117.063;
   1:L PR[91] 10mm/sec FINE;
   1:  PR[GP1:91,1] = PR[GP1:90,1] + 59.525;
   1:  PR[GP1:91,2] = PR[GP1:90,2] + 116.225;
   1:L PR[91] 10mm/sec FINE;
   1:  PR[GP1:91,1] = PR[GP1:90,1] + 59.138;
   1:  PR[GP1:91,2] = PR[GP1:90,2] + 115.339;
   1:L PR[91] 10mm/sec FINE;
   1:  PR[GP1:91,1] = PR[GP1:90,1] + 58.529;
   1:  PR[GP1:91,2] = PR[GP1:90,2] + 111.673;
   1:L PR[91] 10mm/sec FINE;
   1:  PR[GP1:91,1] = PR[GP1:90,1] + 58.284;
   1:  PR[GP1:91,2] = PR[GP1:90,2] + 110.704;
   1:L PR[91] 10mm/sec FINE;
   1:  PR[GP1:91,1] = PR[GP1:90,1] + 58.205;
   1:  PR[GP1:91,2] = PR[GP1:90,2] + 109.741;
   1:L PR[91] 10mm/sec FINE;
   1:  PR[GP1:91,1] = PR[GP1:90,1] + 58.814;
   1:  PR[GP1:91,2] = PR[GP1:90,2] + 106.075;
   1:L PR[91] 10mm/sec FINE;
   1:  PR[GP1:91,1] = PR[GP1:90,1] + 58.897;
   1:  PR[GP1:91,2] = PR[GP1:90,2] + 105.079;
   1:L PR[91] 10mm/sec FINE;
   1:  PR[GP1:91,1] = PR[GP1:90,1] + 59.135;
   1:  PR[GP1:91,2] = PR[GP1:90,2] + 104.133;
   1:L PR[91] 10mm/sec FINE;
   1:  PR[GP1:91,1] = PR[GP1:90,1] + 59.529;
   1:  PR[GP1:91,2] = PR[GP1:90,2] + 103.232;
   1:L PR[91] 10mm/sec FINE;
   1:  PR[GP1:91,1] = PR[GP1:90,1] + 61.292;
   1:  PR[GP1:91,2] = PR[GP1:90,2] + 99.962;
   1:L PR[91] 10mm/sec FINE;
   1:  PR[GP1:91,1] = PR[GP1:90,1] + 61.828;
   1:  PR[GP1:91,2] = PR[GP1:90,2] + 99.137;
   1:L PR[91] 10mm/sec FINE;
   1:  PR[GP1:91,1] = PR[GP1:90,1] + 62.492;
   1:  PR[GP1:91,2] = PR[GP1:90,2] + 98.412;
   1:L PR[91] 10mm/sec FINE;
   1:  PR[GP1:91,1] = PR[GP1:90,1] + 65.219;
   1:  PR[GP1:91,2] = PR[GP1:90,2] + 95.888;
   1:L PR[91] 10mm/sec FINE;
   1:  PR[GP1:91,1] = PR[GP1:90,1] + 65.993;
   1:  PR[GP1:91,2] = PR[GP1:90,2] + 95.282;
   1:L PR[91] 10mm/sec FINE;
   1:  PR[GP1:91,1] = PR[GP1:90,1] + 67.487;
   1:  PR[GP1:91,2] = PR[GP1:90,2] + 94.466;
   1:  PR[GP1:91,3] = PR[GP1:90,3] + 2.900;
   1:L PR[91] 10mm/sec FINE;
   1:  PR[GP1:91,1] = PR[GP1:90,1] + 69.571;
   1:  PR[GP1:91,2] = PR[GP1:90,2] + 93.542;
   1:L PR[91] 10mm/sec FINE;
   1:  PR[GP1:91,1] = PR[GP1:90,1] + 71.180;
   1:  PR[GP1:91,2] = PR[GP1:90,2] + 92.982;
   1:L PR[91] 10mm/sec FINE;
   1:  PR[GP1:91,1] = PR[GP1:90,1] + 72.858;
   1:  PR[GP1:91,2] = PR[GP1:90,2] + 92.693;
   1:L PR[91] 10mm/sec FINE;
   1:  PR[GP1:91,1] = PR[GP1:90,1] + 75.129;
   1:  PR[GP1:91,2] = PR[GP1:90,2] + 92.494;
   1:L PR[91] 10mm/sec FINE;
   1:  PR[GP1:91,1] = PR[GP1:90,1] + 76.833;
   1:  PR[GP1:91,2] = PR[GP1:90,2] + 92.484;
   1:L PR[91] 10mm/sec FINE;
   1:  PR[GP1:91,1] = PR[GP1:90,1] + 78.514;
   1:  PR[GP1:91,2] = PR[GP1:90,2] + 92.754;
   1:L PR[91] 10mm/sec FINE;
   1:  PR[GP1:91,1] = PR[GP1:90,1] + 80.728;
   1:  PR[GP1:91,2] = PR[GP1:90,2] + 93.300;
   1:L PR[91] 10mm/sec FINE;
   1:  PR[GP1:91,1] = PR[GP1:90,1] + 82.342;
   1:  PR[GP1:91,2] = PR[GP1:90,2] + 93.842;
   1:L PR[91] 10mm/sec FINE;
   1:  PR[GP1:91,1] = PR[GP1:90,1] + 83.846;
   1:  PR[GP1:91,2] = PR[GP1:90,2] + 94.642;
   1:L PR[91] 10mm/sec FINE;
   1:  PR[GP1:91,1] = PR[GP1:90,1] + 85.764;
   1:  PR[GP1:91,2] = PR[GP1:90,2] + 95.875;
   1:L PR[91] 10mm/sec FINE;
   1:  PR[GP1:91,1] = PR[GP1:90,1] + 87.116;
   1:  PR[GP1:91,2] = PR[GP1:90,2] + 96.910;
   1:L PR[91] 10mm/sec FINE;
   1:  PR[GP1:91,1] = PR[GP1:90,1] + 88.280;
   1:  PR[GP1:91,2] = PR[GP1:90,2] + 98.153;
   1:L PR[91] 10mm/sec FINE;
   1:  PR[GP1:91,1] = PR[GP1:90,1] + 89.696;
   1:  PR[GP1:91,2] = PR[GP1:90,2] + 99.940;
   1:L PR[91] 10mm/sec FINE;
   1:  PR[GP1:91,1] = PR[GP1:90,1] + 90.640;
   1:  PR[GP1:91,2] = PR[GP1:90,2] + 101.358;
   1:L PR[91] 10mm/sec FINE;
   1:  PR[GP1:91,1] = PR[GP1:90,1] + 91.340;
   1:  PR[GP1:91,2] = PR[GP1:90,2] + 102.911;
   1:L PR[91] 10mm/sec FINE;
   1:  PR[GP1:91,1] = PR[GP1:90,1] + 92.101;
   1:  PR[GP1:91,2] = PR[GP1:90,2] + 105.058;
   1:L PR[91] 10mm/sec FINE;
   1:  PR[GP1:91,1] = PR[GP1:90,1] + 92.544;
   1:  PR[GP1:91,2] = PR[GP1:90,2] + 106.735;
   1:L PR[91] 10mm/sec FINE;
   1:  PR[GP1:91,1] = PR[GP1:90,1] + 93.026;
   1:  PR[GP1:91,2] = PR[GP1:90,2] + 107.850;
   1:L PR[91] 10mm/sec FINE;
   1:  PR[GP1:91,1] = PR[GP1:90,1] + 93.981;
   1:  PR[GP1:91,2] = PR[GP1:90,2] + 108.650;
   1:L PR[91] 10mm/sec FINE;
   1:  PR[GP1:91,1] = PR[GP1:90,1] + 95.171;
   1:  PR[GP1:91,2] = PR[GP1:90,2] + 108.932;
   1:L PR[91] 10mm/sec FINE;
   1:  PR[GP1:91,1] = PR[GP1:90,1] + 95.835;
   1:L PR[91] 10mm/sec FINE;
   1:  PR[GP1:91,1] = PR[GP1:90,1] + 97.025;
   1:  PR[GP1:91,2] = PR[GP1:90,2] + 108.650;
   1:L PR[91] 10mm/sec FINE;
   1:  PR[GP1:91,1] = PR[GP1:90,1] + 97.981;
   1:  PR[GP1:91,2] = PR[GP1:90,2] + 107.850;
   1:L PR[91] 10mm/sec FINE;
   1:  PR[GP1:91,1] = PR[GP1:90,1] + 98.460;
   1:  PR[GP1:91,2] = PR[GP1:90,2] + 106.743;
   1:L PR[91] 10mm/sec FINE;
   1:  PR[GP1:91,1] = PR[GP1:90,1] + 99.232;
   1:  PR[GP1:91,2] = PR[GP1:90,2] + 104.564;
   1:L PR[91] 10mm/sec FINE;
   1:  PR[GP1:91,1] = PR[GP1:90,1] + 99.496;
   1:  PR[GP1:91,2] = PR[GP1:90,2] + 103.442;
   1:L PR[91] 10mm/sec FINE;
   1:  PR[GP1:91,1] = PR[GP1:90,1] + 99.873;
   1:  PR[GP1:91,2] = PR[GP1:90,2] + 102.376;
   1:L PR[91] 10mm/sec FINE;
   1:  PR[GP1:91,1] = PR[GP1:90,1] + 100.361;
   1:  PR[GP1:91,2] = PR[GP1:90,2] + 101.368;
   1:L PR[91] 10mm/sec FINE;
   1:  PR[GP1:91,1] = PR[GP1:90,1] + 101.780;
   1:  PR[GP1:91,2] = PR[GP1:90,2] + 99.576;
   1:L PR[91] 10mm/sec FINE;
   1:  PR[GP1:91,1] = PR[GP1:90,1] + 102.393;
   1:  PR[GP1:91,2] = PR[GP1:90,2] + 98.600;
   1:L PR[91] 10mm/sec FINE;
   1:  PR[GP1:91,1] = PR[GP1:90,1] + 103.095;
   1:  PR[GP1:91,2] = PR[GP1:90,2] + 97.714;
   1:L PR[91] 10mm/sec FINE;
   1:  PR[GP1:91,1] = PR[GP1:90,1] + 103.882;
   1:  PR[GP1:91,2] = PR[GP1:90,2] + 96.918;
   1:L PR[91] 10mm/sec FINE;
   1:  PR[GP1:91,1] = PR[GP1:90,1] + 105.804;
   1:  PR[GP1:91,2] = PR[GP1:90,2] + 95.682;
   1:L PR[91] 10mm/sec FINE;
   1:  PR[GP1:91,1] = PR[GP1:90,1] + 106.700;
   1:  PR[GP1:91,2] = PR[GP1:90,2] + 94.957;
   1:L PR[91] 10mm/sec FINE;
   1:  PR[GP1:91,1] = PR[GP1:90,1] + 107.651;
   1:  PR[GP1:91,2] = PR[GP1:90,2] + 94.345;
   1:L PR[91] 10mm/sec FINE;
   1:  PR[GP1:91,1] = PR[GP1:90,1] + 108.654;
   1:  PR[GP1:91,2] = PR[GP1:90,2] + 93.847;
   1:L PR[91] 10mm/sec FINE;
   1:  PR[GP1:91,1] = PR[GP1:90,1] + 110.873;
   1:  PR[GP1:91,2] = PR[GP1:90,2] + 93.300;
   1:L PR[91] 10mm/sec FINE;
   1:  PR[GP1:91,1] = PR[GP1:90,1] + 111.955;
   1:  PR[GP1:91,2] = PR[GP1:90,2] + 92.903;
   1:L PR[91] 10mm/sec FINE;
   1:  PR[GP1:91,1] = PR[GP1:90,1] + 113.053;
   1:  PR[GP1:91,2] = PR[GP1:90,2] + 92.632;
   1:L PR[91] 10mm/sec FINE;
   1:  PR[GP1:91,1] = PR[GP1:90,1] + 114.163;
   1:  PR[GP1:91,2] = PR[GP1:90,2] + 92.485;
   1:L PR[91] 10mm/sec FINE;
   1:  PR[GP1:91,1] = PR[GP1:90,1] + 116.439;
   1:  PR[GP1:91,2] = PR[GP1:90,2] + 92.685;
   1:L PR[91] 10mm/sec FINE;
   1:  PR[GP1:91,1] = PR[GP1:90,1] + 117.591;
   1:  PR[GP1:91,2] = PR[GP1:90,2] + 92.660;
   1:L PR[91] 10mm/sec FINE;
   1:  PR[GP1:91,1] = PR[GP1:90,1] + 118.718;
   1:  PR[GP1:91,2] = PR[GP1:90,2] + 92.759;
   1:L PR[91] 10mm/sec FINE;
   1:  PR[GP1:91,1] = PR[GP1:90,1] + 119.816;
   1:  PR[GP1:91,2] = PR[GP1:90,2] + 92.979;
   1:L PR[91] 10mm/sec FINE;
   1:  PR[GP1:91,1] = PR[GP1:90,1] + 121.905;
   1:  PR[GP1:91,2] = PR[GP1:90,2] + 93.905;
   1:L PR[91] 10mm/sec FINE;
   1:  PR[GP1:91,1] = PR[GP1:90,1] + 123.003;
   1:  PR[GP1:91,2] = PR[GP1:90,2] + 94.254;
   1:L PR[91] 10mm/sec FINE;
   1:  PR[GP1:91,1] = PR[GP1:90,1] + 124.037;
   1:  PR[GP1:91,2] = PR[GP1:90,2] + 94.713;
   1:L PR[91] 10mm/sec FINE;
   1:  PR[GP1:91,1] = PR[GP1:90,1] + 125.005;
   1:  PR[GP1:91,2] = PR[GP1:90,2] + 95.276;
   1:L PR[91] 10mm/sec FINE;
   1:  PR[GP1:91,1] = PR[GP1:90,1] + 126.682;
   1:  PR[GP1:91,2] = PR[GP1:90,2] + 96.828;
   1:L PR[91] 10mm/sec FINE;
   1:  PR[GP1:91,1] = PR[GP1:90,1] + 127.609;
   1:  PR[GP1:91,2] = PR[GP1:90,2] + 97.514;
   1:L PR[91] 10mm/sec FINE;
   1:  PR[GP1:91,1] = PR[GP1:90,1] + 128.438;
   1:  PR[GP1:91,2] = PR[GP1:90,2] + 98.282;
   1:L PR[91] 10mm/sec FINE;
   1:  PR[GP1:91,1] = PR[GP1:90,1] + 129.171;
   1:  PR[GP1:91,2] = PR[GP1:90,2] + 99.129;
   1:L PR[91] 10mm/sec FINE;
   1:  PR[GP1:91,1] = PR[GP1:90,1] + 130.256;
   1:  PR[GP1:91,2] = PR[GP1:90,2] + 101.141;
   1:L PR[91] 10mm/sec FINE;
   1:  PR[GP1:91,1] = PR[GP1:90,1] + 130.911;
   1:  PR[GP1:91,2] = PR[GP1:90,2] + 102.089;
   1:L PR[91] 10mm/sec FINE;
   1:  PR[GP1:91,1] = PR[GP1:90,1] + 131.448;
   1:  PR[GP1:91,2] = PR[GP1:90,2] + 103.085;
   1:L PR[91] 10mm/sec FINE;
   1:  PR[GP1:91,1] = PR[GP1:90,1] + 131.868;
   1:  PR[GP1:91,2] = PR[GP1:90,2] + 104.123;
   1:L PR[91] 10mm/sec FINE;
   1:  PR[GP1:91,1] = PR[GP1:90,1] + 132.243;
   1:  PR[GP1:91,2] = PR[GP1:90,2] + 106.378;
   1:L PR[91] 10mm/sec FINE;
   1:  PR[GP1:91,1] = PR[GP1:90,1] + 132.555;
   1:  PR[GP1:91,2] = PR[GP1:90,2] + 107.488;
   1:L PR[91] 10mm/sec FINE;
   1:  PR[GP1:91,1] = PR[GP1:90,1] + 132.741;
   1:  PR[GP1:91,2] = PR[GP1:90,2] + 108.603;
   1:L PR[91] 10mm/sec FINE;
   1:  PR[GP1:91,1] = PR[GP1:90,1] + 132.802;
   1:  PR[GP1:91,2] = PR[GP1:90,2] + 109.721;
   1:L PR[91] 10mm/sec FINE;
   1:  PR[GP1:91,1] = PR[GP1:90,1] + 132.428;
   1:  PR[GP1:91,2] = PR[GP1:90,2] + 111.972;
   1:L PR[91] 10mm/sec FINE;
   1:  PR[GP1:91,1] = PR[GP1:90,1] + 132.224;
   1:  PR[GP1:91,2] = PR[GP1:90,2] + 114.025;
   1:L PR[91] 10mm/sec FINE;
   1:  PR[GP1:91,1] = PR[GP1:90,1] + 131.871;
   1:  PR[GP1:91,2] = PR[GP1:90,2] + 115.335;
   1:L PR[91] 10mm/sec FINE;
   1:  PR[GP1:91,1] = PR[GP1:90,1] + 131.633;
   1:  PR[GP1:91,2] = PR[GP1:90,2] + 115.962;
   1:L PR[91] 10mm/sec FINE;
   1:  PR[GP1:91,1] = PR[GP1:90,1] + 129.570;
   1:  PR[GP1:91,2] = PR[GP1:90,2] + 119.786;
   1:L PR[91] 10mm/sec FINE;
   1:  PR[GP1:91,1] = PR[GP1:90,1] + 129.181;
   1:  PR[GP1:91,2] = PR[GP1:90,2] + 120.325;
   1:L PR[91] 10mm/sec FINE;
   1:  PR[GP1:91,1] = PR[GP1:90,1] + 128.272;
   1:  PR[GP1:91,2] = PR[GP1:90,2] + 121.350;
   1:L PR[91] 10mm/sec FINE;
   1:  PR[GP1:91,1] = PR[GP1:90,1] + 126.599;
   1:  PR[GP1:91,2] = PR[GP1:90,2] + 122.898;
   1:L PR[91] 10mm/sec FINE;
   1:  PR[GP1:91,1] = PR[GP1:90,1] + 125.012;
   1:  PR[GP1:91,2] = PR[GP1:90,2] + 124.183;
   1:L PR[91] 10mm/sec FINE;
   1:  PR[GP1:91,1] = PR[GP1:90,1] + 122.931;
   1:  PR[GP1:91,2] = PR[GP1:90,2] + 125.105;
   1:L PR[91] 10mm/sec FINE;
   1:  PR[GP1:91,1] = PR[GP1:90,1] + 121.102;
   1:  PR[GP1:91,2] = PR[GP1:90,2] + 126.063;
   1:L PR[91] 10mm/sec FINE;
   1:  PR[GP1:91,1] = PR[GP1:90,1] + 119.823;
   1:  PR[GP1:91,2] = PR[GP1:90,2] + 126.484;
   1:L PR[91] 10mm/sec FINE;
   1:  PR[GP1:91,1] = PR[GP1:90,1] + 119.158;
   1:  PR[GP1:91,2] = PR[GP1:90,2] + 126.632;
   1:L PR[91] 10mm/sec FINE;
   1:  PR[GP1:91,1] = PR[GP1:90,1] + 114.831;
   1:  PR[GP1:91,2] = PR[GP1:90,2] + 127.010;
   1:L PR[91] 10mm/sec FINE;
   1:  PR[GP1:91,1] = PR[GP1:90,1] + 114.177;
   1:  PR[GP1:91,2] = PR[GP1:90,2] + 126.981;
   1:L PR[91] 10mm/sec FINE;
   1:  PR[GP1:91,1] = PR[GP1:90,1] + 112.811;
   1:  PR[GP1:91,2] = PR[GP1:90,2] + 126.784;
   1:L PR[91] 10mm/sec FINE;
   1:  PR[GP1:91,1] = PR[GP1:90,1] + 110.598;
   1:  PR[GP1:91,2] = PR[GP1:90,2] + 126.238;
   1:L PR[91] 10mm/sec FINE;
   1:  PR[GP1:91,1] = PR[GP1:90,1] + 108.671;
   1:  PR[GP1:91,2] = PR[GP1:90,2] + 125.624;
   1:L PR[91] 10mm/sec FINE;
   1:  PR[GP1:91,1] = PR[GP1:90,1] + 106.739;
   1:  PR[GP1:91,2] = PR[GP1:90,2] + 124.386;
   1:L PR[91] 10mm/sec FINE;
   1:  PR[GP1:91,1] = PR[GP1:90,1] + 104.934;
   1:  PR[GP1:91,2] = PR[GP1:90,2] + 123.383;
   1:L PR[91] 10mm/sec FINE;
   1:  PR[GP1:91,1] = PR[GP1:90,1] + 103.888;
   1:  PR[GP1:91,2] = PR[GP1:90,2] + 122.553;
   1:L PR[91] 10mm/sec FINE;
   1:  PR[GP1:91,1] = PR[GP1:90,1] + 103.391;
   1:  PR[GP1:91,2] = PR[GP1:90,2] + 122.071;
   1:L PR[91] 10mm/sec FINE;
   1:  PR[GP1:91,1] = PR[GP1:90,1] + 100.697;
   1:  PR[GP1:91,2] = PR[GP1:90,2] + 118.663;
   1:L PR[91] 10mm/sec FINE;
   1:  PR[GP1:91,1] = PR[GP1:90,1] + 100.367;
   1:  PR[GP1:91,2] = PR[GP1:90,2] + 118.110;
   1:L PR[91] 10mm/sec FINE;
   1:  PR[GP1:91,1] = PR[GP1:90,1] + 99.777;
   1:  PR[GP1:91,2] = PR[GP1:90,2] + 116.851;
   1:L PR[91] 10mm/sec FINE;
   1:  PR[GP1:91,1] = PR[GP1:90,1] + 99.017;
   1:  PR[GP1:91,2] = PR[GP1:90,2] + 114.704;
   1:L PR[91] 10mm/sec FINE;
   1:  PR[GP1:91,1] = PR[GP1:90,1] + 98.462;
   1:  PR[GP1:91,2] = PR[GP1:90,2] + 112.728;
   1:L PR[91] 10mm/sec FINE;
   1:  PR[GP1:91,1] = PR[GP1:90,1] + 97.981;
   1:  PR[GP1:91,2] = PR[GP1:90,2] + 111.615;
   1:L PR[91] 10mm/sec FINE;
   1:  PR[GP1:91,1] = PR[GP1:90,1] + 97.025;
   1:  PR[GP1:91,2] = PR[GP1:90,2] + 110.814;
   1:L PR[91] 10mm/sec FINE;
   1:  PR[GP1:91,1] = PR[GP1:90,1] + 95.835;
   1:  PR[GP1:91,2] = PR[GP1:90,2] + 110.532;
   1:L PR[91] 10mm/sec FINE;
   1:  PR[GP1:91,1] = PR[GP1:90,1] + 95.171;
   1:L PR[91] 10mm/sec FINE;
   1:  PR[GP1:91,1] = PR[GP1:90,1] + 93.981;
   1:  PR[GP1:91,2] = PR[GP1:90,2] + 110.814;
   1:L PR[91] 10mm/sec FINE;
   1:  PR[GP1:91,1] = PR[GP1:90,1] + 93.026;
   1:  PR[GP1:91,2] = PR[GP1:90,2] + 111.615;
   1:L PR[91] 10mm/sec FINE;
   1:  PR[GP1:91,1] = PR[GP1:90,1] + 92.547;
   1:  PR[GP1:91,2] = PR[GP1:90,2] + 112.721;
   1:L PR[91] 10mm/sec FINE;
   1:  PR[GP1:91,1] = PR[GP1:90,1] + 91.776;
   1:  PR[GP1:91,2] = PR[GP1:90,2] + 114.898;
   1:L PR[91] 10mm/sec FINE;
   1:  PR[GP1:91,1] = PR[GP1:90,1] + 91.336;
   1:  PR[GP1:91,2] = PR[GP1:90,2] + 116.561;
   1:L PR[91] 10mm/sec FINE;
   1:  PR[GP1:91,1] = PR[GP1:90,1] + 90.644;
   1:  PR[GP1:91,2] = PR[GP1:90,2] + 118.099;
   1:L PR[91] 10mm/sec FINE;
   1:  PR[GP1:91,1] = PR[GP1:90,1] + 89.228;
   1:  PR[GP1:91,2] = PR[GP1:90,2] + 119.886;
   1:L PR[91] 10mm/sec FINE;
   1:  PR[GP1:91,1] = PR[GP1:90,1] + 88.275;
   1:  PR[GP1:91,2] = PR[GP1:90,2] + 121.317;
   1:L PR[91] 10mm/sec FINE;
   1:  PR[GP1:91,1] = PR[GP1:90,1] + 87.122;
   1:  PR[GP1:91,2] = PR[GP1:90,2] + 122.548;
   1:L PR[91] 10mm/sec FINE;
   1:  PR[GP1:91,1] = PR[GP1:90,1] + 85.204;
   1:  PR[GP1:91,2] = PR[GP1:90,2] + 123.781;
   1:L PR[91] 10mm/sec FINE;
   1:  PR[GP1:91,1] = PR[GP1:90,1] + 83.839;
   1:  PR[GP1:91,2] = PR[GP1:90,2] + 124.826;
   1:L PR[91] 10mm/sec FINE;
   1:  PR[GP1:91,1] = PR[GP1:90,1] + 82.350;
   1:  PR[GP1:91,2] = PR[GP1:90,2] + 125.618;
   1:L PR[91] 10mm/sec FINE;
   1:  PR[GP1:91,1] = PR[GP1:90,1] + 80.136;
   1:  PR[GP1:91,2] = PR[GP1:90,2] + 126.164;
   1:L PR[91] 10mm/sec FINE;
   1:  PR[GP1:91,1] = PR[GP1:90,1] + 78.506;
   1:  PR[GP1:91,2] = PR[GP1:90,2] + 126.712;
   1:L PR[91] 10mm/sec FINE;
   1:  PR[GP1:91,1] = PR[GP1:90,1] + 76.841;
   1:  PR[GP1:91,2] = PR[GP1:90,2] + 126.979;
   1:L PR[91] 10mm/sec FINE;
   1:  PR[GP1:91,1] = PR[GP1:90,1] + 74.570;
   1:  PR[GP1:91,2] = PR[GP1:90,2] + 126.779;
   1:L PR[91] 10mm/sec FINE;
   1:  PR[GP1:91,1] = PR[GP1:90,1] + 72.850;
   1:  PR[GP1:91,2] = PR[GP1:90,2] + 126.770;
   1:L PR[91] 10mm/sec FINE;
   1:  PR[GP1:91,1] = PR[GP1:90,1] + 71.188;
   1:  PR[GP1:91,2] = PR[GP1:90,2] + 126.484;
   1:L PR[91] 10mm/sec FINE;
   1:  PR[GP1:91,1] = PR[GP1:90,1] + 69.104;
   1:  PR[GP1:91,2] = PR[GP1:90,2] + 125.560;
   1:L PR[91] 10mm/sec FINE;
   1:  PR[GP1:91,1] = PR[GP1:90,1] + 67.480;
   1:  PR[GP1:91,2] = PR[GP1:90,2] + 124.995;
   1:L PR[91] 10mm/sec FINE;
   1:  PR[GP1:91,1] = PR[GP1:90,1] + 65.999;
   1:  PR[GP1:91,2] = PR[GP1:90,2] + 124.186;
   1:L PR[91] 10mm/sec FINE;
   1:  PR[GP1:91,1] = PR[GP1:90,1] + 64.326;
   1:  PR[GP1:91,2] = PR[GP1:90,2] + 122.637;
   1:L PR[91] 10mm/sec FINE;
   1:  PR[GP1:91,1] = PR[GP1:90,1] + 62.972;
   1:  PR[GP1:91,2] = PR[GP1:90,2] + 121.577;
   1:L PR[91] 10mm/sec FINE;
   1:  PR[GP1:91,1] = PR[GP1:90,1] + 61.833;
   1:  PR[GP1:91,2] = PR[GP1:90,2] + 120.333;
   1:L PR[91] 10mm/sec FINE;
   1:  PR[GP1:91,1] = PR[GP1:90,1] + 60.751;
   1:  PR[GP1:91,2] = PR[GP1:90,2] + 118.326;
   1:L PR[91] 10mm/sec FINE;
   1:  PR[GP1:91,1] = PR[GP1:90,1] + 59.814;
   1:  PR[GP1:91,2] = PR[GP1:90,2] + 116.884;
   1:L PR[91] 10mm/sec FINE;
   1:  PR[GP1:91,1] = PR[GP1:90,1] + 59.138;
   1:  PR[GP1:91,2] = PR[GP1:90,2] + 115.338;
   1:L PR[91] 10mm/sec FINE;
   1:  PR[GP1:91,1] = PR[GP1:90,1] + 58.764;
   1:  PR[GP1:91,2] = PR[GP1:90,2] + 113.089;
   1:L PR[91] 10mm/sec FINE;
   1:  PR[GP1:91,1] = PR[GP1:90,1] + 58.343;
   1:  PR[GP1:91,2] = PR[GP1:90,2] + 111.421;
   1:L PR[91] 10mm/sec FINE;
   1:  PR[GP1:91,1] = PR[GP1:90,1] + 58.205;
   1:  PR[GP1:91,2] = PR[GP1:90,2] + 109.741;
   1:L PR[91] 10mm/sec FINE;
   1:  PR[GP1:91,1] = PR[GP1:90,1] + 58.579;
   1:  PR[GP1:91,2] = PR[GP1:90,2] + 107.491;
   1:L PR[91] 10mm/sec FINE;
   1:  PR[GP1:91,1] = PR[GP1:90,1] + 58.720;
   1:  PR[GP1:91,2] = PR[GP1:90,2] + 105.777;
   1:L PR[91] 10mm/sec FINE;
   1:  PR[GP1:91,1] = PR[GP1:90,1] + 59.135;
   1:  PR[GP1:91,2] = PR[GP1:90,2] + 104.134;
   1:L PR[91] 10mm/sec FINE;
   1:  PR[GP1:91,1] = PR[GP1:90,1] + 59.817;
   1:  PR[GP1:91,2] = PR[GP1:90,2] + 102.573;
   1:L PR[91] 10mm/sec FINE;
   1:  PR[GP1:91,1] = PR[GP1:90,1] + 60.899;
   1:  PR[GP1:91,2] = PR[GP1:90,2] + 100.566;
   1:L PR[91] 10mm/sec FINE;
   1:  PR[GP1:91,1] = PR[GP1:90,1] + 61.828;
   1:  PR[GP1:91,2] = PR[GP1:90,2] + 99.138;
   1:L PR[91] 10mm/sec FINE;
   1:  PR[GP1:91,1] = PR[GP1:90,1] + 62.978;
   1:  PR[GP1:91,2] = PR[GP1:90,2] + 97.882;
   1:L PR[91] 10mm/sec FINE;
   1:  PR[GP1:91,1] = PR[GP1:90,1] + 64.651;
   1:  PR[GP1:91,2] = PR[GP1:90,2] + 96.333;
   1:L PR[91] 10mm/sec FINE;
   1:  PR[GP1:91,1] = PR[GP1:90,1] + 65.992;
   1:  PR[GP1:91,2] = PR[GP1:90,2] + 95.282;
   1:L PR[91] 10mm/sec FINE;
   1:  PR[GP1:91,1] = PR[GP1:90,1] + 68.118;
   1:  PR[GP1:91,2] = PR[GP1:90,2] + 94.121;
   1:  PR[GP1:91,3] = PR[GP1:90,3] + 3.900;
   1:L PR[91] 10mm/sec FINE;
   1:  PR[GP1:91,1] = PR[GP1:90,1] + 68.890;
   1:  PR[GP1:91,2] = PR[GP1:90,2] + 93.779;
   1:L PR[91] 10mm/sec FINE;
   1:  PR[GP1:91,1] = PR[GP1:90,1] + 71.179;
   1:  PR[GP1:91,2] = PR[GP1:90,2] + 92.982;
   1:L PR[91] 10mm/sec FINE;
   1:  PR[GP1:91,1] = PR[GP1:90,1] + 73.567;
   1:  PR[GP1:91,2] = PR[GP1:90,2] + 92.571;
   1:L PR[91] 10mm/sec FINE;
   1:  PR[GP1:91,1] = PR[GP1:90,1] + 74.408;
   1:  PR[GP1:91,2] = PR[GP1:90,2] + 92.497;
   1:L PR[91] 10mm/sec FINE;
   1:  PR[GP1:91,1] = PR[GP1:90,1] + 76.831;
   1:  PR[GP1:91,2] = PR[GP1:90,2] + 92.484;
   1:L PR[91] 10mm/sec FINE;
   1:  PR[GP1:91,1] = PR[GP1:90,1] + 79.224;
   1:  PR[GP1:91,2] = PR[GP1:90,2] + 92.868;
   1:L PR[91] 10mm/sec FINE;
   1:  PR[GP1:91,1] = PR[GP1:90,1] + 80.044;
   1:  PR[GP1:91,2] = PR[GP1:90,2] + 93.070;
   1:L PR[91] 10mm/sec FINE;
   1:  PR[GP1:91,1] = PR[GP1:90,1] + 82.341;
   1:  PR[GP1:91,2] = PR[GP1:90,2] + 93.842;
   1:L PR[91] 10mm/sec FINE;
   1:  PR[GP1:91,1] = PR[GP1:90,1] + 84.481;
   1:  PR[GP1:91,2] = PR[GP1:90,2] + 94.979;
   1:L PR[91] 10mm/sec FINE;
   1:  PR[GP1:91,1] = PR[GP1:90,1] + 85.191;
   1:  PR[GP1:91,2] = PR[GP1:90,2] + 95.436;
   1:L PR[91] 10mm/sec FINE;
   1:  PR[GP1:91,1] = PR[GP1:90,1] + 87.115;
   1:  PR[GP1:91,2] = PR[GP1:90,2] + 96.909;
   1:L PR[91] 10mm/sec FINE;
   1:  PR[GP1:91,1] = PR[GP1:90,1] + 88.772;
   1:  PR[GP1:91,2] = PR[GP1:90,2] + 98.678;
   1:L PR[91] 10mm/sec FINE;
   1:  PR[GP1:91,1] = PR[GP1:90,1] + 89.296;
   1:  PR[GP1:91,2] = PR[GP1:90,2] + 99.340;
   1:L PR[91] 10mm/sec FINE;
   1:  PR[GP1:91,1] = PR[GP1:90,1] + 90.640;
   1:  PR[GP1:91,2] = PR[GP1:90,2] + 101.357;
   1:L PR[91] 10mm/sec FINE;
   1:  PR[GP1:91,1] = PR[GP1:90,1] + 91.635;
   1:  PR[GP1:91,2] = PR[GP1:90,2] + 103.567;
   1:L PR[91] 10mm/sec FINE;
   1:  PR[GP1:91,1] = PR[GP1:90,1] + 91.917;
   1:  PR[GP1:91,2] = PR[GP1:90,2] + 104.362;
   1:L PR[91] 10mm/sec FINE;
   1:  PR[GP1:91,1] = PR[GP1:90,1] + 92.544;
   1:  PR[GP1:91,2] = PR[GP1:90,2] + 106.735;
   1:L PR[91] 10mm/sec FINE;
   1:  PR[GP1:91,1] = PR[GP1:90,1] + 93.026;
   1:  PR[GP1:91,2] = PR[GP1:90,2] + 107.850;
   1:L PR[91] 10mm/sec FINE;
   1:  PR[GP1:91,1] = PR[GP1:90,1] + 93.981;
   1:  PR[GP1:91,2] = PR[GP1:90,2] + 108.650;
   1:L PR[91] 10mm/sec FINE;
   1:  PR[GP1:91,1] = PR[GP1:90,1] + 95.171;
   1:  PR[GP1:91,2] = PR[GP1:90,2] + 108.932;
   1:L PR[91] 10mm/sec FINE;
   1:  PR[GP1:91,1] = PR[GP1:90,1] + 95.835;
   1:L PR[91] 10mm/sec FINE;
   1:  PR[GP1:91,1] = PR[GP1:90,1] + 97.025;
   1:  PR[GP1:91,2] = PR[GP1:90,2] + 108.650;
   1:L PR[91] 10mm/sec FINE;
   1:  PR[GP1:91,1] = PR[GP1:90,1] + 97.981;
   1:  PR[GP1:91,2] = PR[GP1:90,2] + 107.850;
   1:L PR[91] 10mm/sec FINE;
   1:  PR[GP1:91,1] = PR[GP1:90,1] + 98.460;
   1:  PR[GP1:91,2] = PR[GP1:90,2] + 106.743;
   1:L PR[91] 10mm/sec FINE;
   1:  PR[GP1:91,1] = PR[GP1:90,1] + 98.753;
   1:  PR[GP1:91,2] = PR[GP1:90,2] + 105.915;
   1:L PR[91] 10mm/sec FINE;
   1:  PR[GP1:91,1] = PR[GP1:90,1] + 99.126;
   1:  PR[GP1:91,2] = PR[GP1:90,2] + 104.326;
   1:L PR[91] 10mm/sec FINE;
   1:  PR[GP1:91,1] = PR[GP1:90,1] + 99.665;
   1:  PR[GP1:91,2] = PR[GP1:90,2] + 102.807;
   1:L PR[91] 10mm/sec FINE;
   1:  PR[GP1:91,1] = PR[GP1:90,1] + 100.361;
   1:  PR[GP1:91,2] = PR[GP1:90,2] + 101.367;
   1:L PR[91] 10mm/sec FINE;
   1:  PR[GP1:91,1] = PR[GP1:90,1] + 100.889;
   1:  PR[GP1:91,2] = PR[GP1:90,2] + 100.700;
   1:L PR[91] 10mm/sec FINE;
   1:  PR[GP1:91,1] = PR[GP1:90,1] + 101.757;
   1:  PR[GP1:91,2] = PR[GP1:90,2] + 99.317;
   1:L PR[91] 10mm/sec FINE;
   1:  PR[GP1:91,1] = PR[GP1:90,1] + 102.758;
   1:  PR[GP1:91,2] = PR[GP1:90,2] + 98.054;
   1:L PR[91] 10mm/sec FINE;
   1:  PR[GP1:91,1] = PR[GP1:90,1] + 103.883;
   1:  PR[GP1:91,2] = PR[GP1:90,2] + 96.917;
   1:L PR[91] 10mm/sec FINE;
   1:  PR[GP1:91,1] = PR[GP1:90,1] + 104.598;
   1:  PR[GP1:91,2] = PR[GP1:90,2] + 96.457;
   1:L PR[91] 10mm/sec FINE;
   1:  PR[GP1:91,1] = PR[GP1:90,1] + 105.867;
   1:  PR[GP1:91,2] = PR[GP1:90,2] + 95.429;
   1:L PR[91] 10mm/sec FINE;
   1:  PR[GP1:91,1] = PR[GP1:90,1] + 107.222;
   1:  PR[GP1:91,2] = PR[GP1:90,2] + 94.558;
   1:L PR[91] 10mm/sec FINE;
   1:  PR[GP1:91,1] = PR[GP1:90,1] + 108.655;
   1:  PR[GP1:91,2] = PR[GP1:90,2] + 93.846;
   1:L PR[91] 10mm/sec FINE;
   1:  PR[GP1:91,1] = PR[GP1:90,1] + 109.480;
   1:  PR[GP1:91,2] = PR[GP1:90,2] + 93.643;
   1:L PR[91] 10mm/sec FINE;
   1:  PR[GP1:91,1] = PR[GP1:90,1] + 111.014;
   1:  PR[GP1:91,2] = PR[GP1:90,2] + 93.081;
   1:L PR[91] 10mm/sec FINE;
   1:  PR[GP1:91,1] = PR[GP1:90,1] + 112.578;
   1:  PR[GP1:91,2] = PR[GP1:90,2] + 92.695;
   1:L PR[91] 10mm/sec FINE;
   1:  PR[GP1:91,1] = PR[GP1:90,1] + 114.164;
   1:  PR[GP1:91,2] = PR[GP1:90,2] + 92.485;
   1:L PR[91] 10mm/sec FINE;
   1:  PR[GP1:91,1] = PR[GP1:90,1] + 115.011;
   1:  PR[GP1:91,2] = PR[GP1:90,2] + 92.559;
   1:L PR[91] 10mm/sec FINE;
   1:  PR[GP1:91,1] = PR[GP1:90,1] + 116.643;
   1:  PR[GP1:91,2] = PR[GP1:90,2] + 92.524;
   1:L PR[91] 10mm/sec FINE;
   1:  PR[GP1:91,1] = PR[GP1:90,1] + 118.248;
   1:  PR[GP1:91,2] = PR[GP1:90,2] + 92.665;
   1:L PR[91] 10mm/sec FINE;
   1:  PR[GP1:91,1] = PR[GP1:90,1] + 119.817;
   1:  PR[GP1:91,2] = PR[GP1:90,2] + 92.980;
   1:L PR[91] 10mm/sec FINE;
   1:  PR[GP1:91,1] = PR[GP1:90,1] + 120.594;
   1:  PR[GP1:91,2] = PR[GP1:90,2] + 93.324;
   1:L PR[91] 10mm/sec FINE;
   1:  PR[GP1:91,1] = PR[GP1:90,1] + 122.151;
   1:  PR[GP1:91,2] = PR[GP1:90,2] + 93.819;
   1:L PR[91] 10mm/sec FINE;
   1:  PR[GP1:91,1] = PR[GP1:90,1] + 123.623;
   1:  PR[GP1:91,2] = PR[GP1:90,2] + 94.472;
   1:L PR[91] 10mm/sec FINE;
   1:  PR[GP1:91,1] = PR[GP1:90,1] + 125.006;
   1:  PR[GP1:91,2] = PR[GP1:90,2] + 95.277;
   1:L PR[91] 10mm/sec FINE;
   1:  PR[GP1:91,1] = PR[GP1:90,1] + 125.630;
   1:  PR[GP1:91,2] = PR[GP1:90,2] + 95.854;
   1:L PR[91] 10mm/sec FINE;
   1:  PR[GP1:91,1] = PR[GP1:90,1] + 126.942;
   1:  PR[GP1:91,2] = PR[GP1:90,2] + 96.826;
   1:L PR[91] 10mm/sec FINE;
   1:  PR[GP1:91,1] = PR[GP1:90,1] + 128.125;
   1:  PR[GP1:91,2] = PR[GP1:90,2] + 97.920;
   1:L PR[91] 10mm/sec FINE;
   1:  PR[GP1:91,1] = PR[GP1:90,1] + 129.172;
   1:  PR[GP1:91,2] = PR[GP1:90,2] + 99.130;
   1:L PR[91] 10mm/sec FINE;
   1:  PR[GP1:91,1] = PR[GP1:90,1] + 129.576;
   1:  PR[GP1:91,2] = PR[GP1:90,2] + 99.878;
   1:L PR[91] 10mm/sec FINE;
   1:  PR[GP1:91,1] = PR[GP1:90,1] + 130.504;
   1:  PR[GP1:91,2] = PR[GP1:90,2] + 101.222;
   1:L PR[91] 10mm/sec FINE;
   1:  PR[GP1:91,1] = PR[GP1:90,1] + 131.268;
   1:  PR[GP1:91,2] = PR[GP1:90,2] + 102.640;
   1:L PR[91] 10mm/sec FINE;
   1:  PR[GP1:91,1] = PR[GP1:90,1] + 131.868;
   1:  PR[GP1:91,2] = PR[GP1:90,2] + 104.123;
   1:L PR[91] 10mm/sec FINE;
   1:  PR[GP1:91,1] = PR[GP1:90,1] + 132.007;
   1:  PR[GP1:91,2] = PR[GP1:90,2] + 104.962;
   1:L PR[91] 10mm/sec FINE;
   1:  PR[GP1:91,1] = PR[GP1:90,1] + 132.450;
   1:  PR[GP1:91,2] = PR[GP1:90,2] + 106.534;
   1:L PR[91] 10mm/sec FINE;
   1:  PR[GP1:91,1] = PR[GP1:90,1] + 132.715;
   1:  PR[GP1:91,2] = PR[GP1:90,2] + 108.124;
   1:L PR[91] 10mm/sec FINE;
   1:  PR[GP1:91,1] = PR[GP1:90,1] + 132.802;
   1:  PR[GP1:91,2] = PR[GP1:90,2] + 109.721;
   1:L PR[91] 10mm/sec FINE;
   1:  PR[GP1:91,1] = PR[GP1:90,1] + 132.664;
   1:  PR[GP1:91,2] = PR[GP1:90,2] + 110.556;
   1:L PR[91] 10mm/sec FINE;
   1:  PR[GP1:91,1] = PR[GP1:90,1] + 132.375;
   1:  PR[GP1:91,2] = PR[GP1:90,2] + 113.468;
   1:L PR[91] 10mm/sec FINE;
   1:  PR[GP1:91,1] = PR[GP1:90,1] + 131.871;
   1:  PR[GP1:91,2] = PR[GP1:90,2] + 115.334;
   1:L PR[91] 10mm/sec FINE;
   1:  PR[GP1:91,1] = PR[GP1:90,1] + 131.531;
   1:  PR[GP1:91,2] = PR[GP1:90,2] + 116.231;
   1:L PR[91] 10mm/sec FINE;
   1:  PR[GP1:91,1] = PR[GP1:90,1] + 129.739;
   1:  PR[GP1:91,2] = PR[GP1:90,2] + 119.553;
   1:L PR[91] 10mm/sec FINE;
   1:  PR[GP1:91,1] = PR[GP1:90,1] + 129.182;
   1:  PR[GP1:91,2] = PR[GP1:90,2] + 120.324;
   1:L PR[91] 10mm/sec FINE;
   1:  PR[GP1:91,1] = PR[GP1:90,1] + 127.889;
   1:  PR[GP1:91,2] = PR[GP1:90,2] + 121.782;
   1:L PR[91] 10mm/sec FINE;
   1:  PR[GP1:91,1] = PR[GP1:90,1] + 127.269;
   1:  PR[GP1:91,2] = PR[GP1:90,2] + 122.355;
   1:L PR[91] 10mm/sec FINE;
   1:  PR[GP1:91,1] = PR[GP1:90,1] + 125.010;
   1:  PR[GP1:91,2] = PR[GP1:90,2] + 124.184;
   1:L PR[91] 10mm/sec FINE;
   1:  PR[GP1:91,1] = PR[GP1:90,1] + 124.241;
   1:  PR[GP1:91,2] = PR[GP1:90,2] + 124.524;
   1:L PR[91] 10mm/sec FINE;
   1:  PR[GP1:91,1] = PR[GP1:90,1] + 121.647;
   1:  PR[GP1:91,2] = PR[GP1:90,2] + 125.884;
   1:L PR[91] 10mm/sec FINE;
   1:  PR[GP1:91,1] = PR[GP1:90,1] + 119.825;
   1:  PR[GP1:91,2] = PR[GP1:90,2] + 126.483;
   1:L PR[91] 10mm/sec FINE;
   1:  PR[GP1:91,1] = PR[GP1:90,1] + 118.873;
   1:  PR[GP1:91,2] = PR[GP1:90,2] + 126.695;
   1:L PR[91] 10mm/sec FINE;
   1:  PR[GP1:91,1] = PR[GP1:90,1] + 115.114;
   1:  PR[GP1:91,2] = PR[GP1:90,2] + 127.023;
   1:L PR[91] 10mm/sec FINE;
   1:  PR[GP1:91,1] = PR[GP1:90,1] + 114.178;
   1:  PR[GP1:91,2] = PR[GP1:90,2] + 126.981;
   1:L PR[91] 10mm/sec FINE;
   1:  PR[GP1:91,1] = PR[GP1:90,1] + 112.236;
   1:  PR[GP1:91,2] = PR[GP1:90,2] + 126.700;
   1:L PR[91] 10mm/sec FINE;
   1:  PR[GP1:91,1] = PR[GP1:90,1] + 111.416;
   1:  PR[GP1:91,2] = PR[GP1:90,2] + 126.498;
   1:L PR[91] 10mm/sec FINE;
   1:  PR[GP1:91,1] = PR[GP1:90,1] + 108.671;
   1:  PR[GP1:91,2] = PR[GP1:90,2] + 125.624;
   1:L PR[91] 10mm/sec FINE;
   1:  PR[GP1:91,1] = PR[GP1:90,1] + 107.940;
   1:  PR[GP1:91,2] = PR[GP1:90,2] + 125.159;
   1:L PR[91] 10mm/sec FINE;
   1:  PR[GP1:91,1] = PR[GP1:90,1] + 105.379;
   1:  PR[GP1:91,2] = PR[GP1:90,2] + 123.737;
   1:L PR[91] 10mm/sec FINE;
   1:  PR[GP1:91,1] = PR[GP1:90,1] + 103.889;
   1:  PR[GP1:91,2] = PR[GP1:90,2] + 122.553;
   1:L PR[91] 10mm/sec FINE;
   1:  PR[GP1:91,1] = PR[GP1:90,1] + 103.178;
   1:  PR[GP1:91,2] = PR[GP1:90,2] + 121.865;
   1:L PR[91] 10mm/sec FINE;
   1:  PR[GP1:91,1] = PR[GP1:90,1] + 100.840;
   1:  PR[GP1:91,2] = PR[GP1:90,2] + 118.903;
   1:L PR[91] 10mm/sec FINE;
   1:  PR[GP1:91,1] = PR[GP1:90,1] + 100.368;
   1:  PR[GP1:91,2] = PR[GP1:90,2] + 118.111;
   1:L PR[91] 10mm/sec FINE;
   1:  PR[GP1:91,1] = PR[GP1:90,1] + 99.529;
   1:  PR[GP1:91,2] = PR[GP1:90,2] + 116.320;
   1:L PR[91] 10mm/sec FINE;
   1:  PR[GP1:91,1] = PR[GP1:90,1] + 99.247;
   1:  PR[GP1:91,2] = PR[GP1:90,2] + 115.525;
   1:L PR[91] 10mm/sec FINE;
   1:  PR[GP1:91,1] = PR[GP1:90,1] + 98.462;
   1:  PR[GP1:91,2] = PR[GP1:90,2] + 112.728;
   1:L PR[91] 10mm/sec FINE;
   1:  PR[GP1:91,1] = PR[GP1:90,1] + 97.981;
   1:  PR[GP1:91,2] = PR[GP1:90,2] + 111.615;
   1:L PR[91] 10mm/sec FINE;
   1:  PR[GP1:91,1] = PR[GP1:90,1] + 97.025;
   1:  PR[GP1:91,2] = PR[GP1:90,2] + 110.814;
   1:L PR[91] 10mm/sec FINE;
   1:  PR[GP1:91,1] = PR[GP1:90,1] + 95.835;
   1:  PR[GP1:91,2] = PR[GP1:90,2] + 110.532;
   1:L PR[91] 10mm/sec FINE;
   1:  PR[GP1:91,1] = PR[GP1:90,1] + 95.171;
   1:L PR[91] 10mm/sec FINE;
   1:  PR[GP1:91,1] = PR[GP1:90,1] + 93.981;
   1:  PR[GP1:91,2] = PR[GP1:90,2] + 110.814;
   1:L PR[91] 10mm/sec FINE;
   1:  PR[GP1:91,1] = PR[GP1:90,1] + 93.026;
   1:  PR[GP1:91,2] = PR[GP1:90,2] + 111.615;
   1:L PR[91] 10mm/sec FINE;
   1:  PR[GP1:91,1] = PR[GP1:90,1] + 92.547;
   1:  PR[GP1:91,2] = PR[GP1:90,2] + 112.721;
   1:L PR[91] 10mm/sec FINE;
   1:  PR[GP1:91,1] = PR[GP1:90,1] + 92.255;
   1:  PR[GP1:91,2] = PR[GP1:90,2] + 113.547;
   1:L PR[91] 10mm/sec FINE;
   1:  PR[GP1:91,1] = PR[GP1:90,1] + 91.631;
   1:  PR[GP1:91,2] = PR[GP1:90,2] + 115.906;
   1:L PR[91] 10mm/sec FINE;
   1:  PR[GP1:91,1] = PR[GP1:90,1] + 90.643;
   1:  PR[GP1:91,2] = PR[GP1:90,2] + 118.100;
   1:L PR[91] 10mm/sec FINE;
   1:  PR[GP1:91,1] = PR[GP1:90,1] + 90.119;
   1:  PR[GP1:91,2] = PR[GP1:90,2] + 118.762;
   1:L PR[91] 10mm/sec FINE;
   1:  PR[GP1:91,1] = PR[GP1:90,1] + 88.766;
   1:  PR[GP1:91,2] = PR[GP1:90,2] + 120.792;
   1:L PR[91] 10mm/sec FINE;
   1:  PR[GP1:91,1] = PR[GP1:90,1] + 87.121;
   1:  PR[GP1:91,2] = PR[GP1:90,2] + 122.549;
   1:L PR[91] 10mm/sec FINE;
   1:  PR[GP1:91,1] = PR[GP1:90,1] + 86.411;
   1:  PR[GP1:91,2] = PR[GP1:90,2] + 123.006;
   1:L PR[91] 10mm/sec FINE;
   1:  PR[GP1:91,1] = PR[GP1:90,1] + 84.474;
   1:  PR[GP1:91,2] = PR[GP1:90,2] + 124.489;
   1:L PR[91] 10mm/sec FINE;
   1:  PR[GP1:91,1] = PR[GP1:90,1] + 82.349;
   1:  PR[GP1:91,2] = PR[GP1:90,2] + 125.619;
   1:L PR[91] 10mm/sec FINE;
   1:  PR[GP1:91,1] = PR[GP1:90,1] + 81.529;
   1:  PR[GP1:91,2] = PR[GP1:90,2] + 125.821;
   1:L PR[91] 10mm/sec FINE;
   1:  PR[GP1:91,1] = PR[GP1:90,1] + 79.216;
   1:  PR[GP1:91,2] = PR[GP1:90,2] + 126.598;
   1:L PR[91] 10mm/sec FINE;
   1:  PR[GP1:91,1] = PR[GP1:90,1] + 76.840;
   1:  PR[GP1:91,2] = PR[GP1:90,2] + 126.979;
   1:L PR[91] 10mm/sec FINE;
   1:  PR[GP1:91,1] = PR[GP1:90,1] + 75.998;
   1:  PR[GP1:91,2] = PR[GP1:90,2] + 126.905;
   1:L PR[91] 10mm/sec FINE;
   1:  PR[GP1:91,1] = PR[GP1:90,1] + 73.559;
   1:  PR[GP1:91,2] = PR[GP1:90,2] + 126.892;
   1:L PR[91] 10mm/sec FINE;
   1:  PR[GP1:91,1] = PR[GP1:90,1] + 71.187;
   1:  PR[GP1:91,2] = PR[GP1:90,2] + 126.484;
   1:L PR[91] 10mm/sec FINE;
   1:  PR[GP1:91,1] = PR[GP1:90,1] + 70.415;
   1:  PR[GP1:91,2] = PR[GP1:90,2] + 126.141;
   1:L PR[91] 10mm/sec FINE;
   1:  PR[GP1:91,1] = PR[GP1:90,1] + 68.111;
   1:  PR[GP1:91,2] = PR[GP1:90,2] + 125.339;
   1:L PR[91] 10mm/sec FINE;
   1:  PR[GP1:91,1] = PR[GP1:90,1] + 65.998;
   1:  PR[GP1:91,2] = PR[GP1:90,2] + 124.186;
   1:L PR[91] 10mm/sec FINE;
   1:  PR[GP1:91,1] = PR[GP1:90,1] + 65.379;
   1:  PR[GP1:91,2] = PR[GP1:90,2] + 123.612;
   1:L PR[91] 10mm/sec FINE;
   1:  PR[GP1:91,1] = PR[GP1:90,1] + 63.458;
   1:  PR[GP1:91,2] = PR[GP1:90,2] + 122.107;
   1:L PR[91] 10mm/sec FINE;
   1:  PR[GP1:91,1] = PR[GP1:90,1] + 61.833;
   1:  PR[GP1:91,2] = PR[GP1:90,2] + 120.332;
   1:L PR[91] 10mm/sec FINE;
   1:  PR[GP1:91,1] = PR[GP1:90,1] + 61.432;
   1:  PR[GP1:91,2] = PR[GP1:90,2] + 119.589;
   1:L PR[91] 10mm/sec FINE;
   1:  PR[GP1:91,1] = PR[GP1:90,1] + 60.102;
   1:  PR[GP1:91,2] = PR[GP1:90,2] + 117.543;
   1:L PR[91] 10mm/sec FINE;
   1:  PR[GP1:91,1] = PR[GP1:90,1] + 59.138;
   1:  PR[GP1:91,2] = PR[GP1:90,2] + 115.338;
   1:L PR[91] 10mm/sec FINE;
   1:  PR[GP1:91,1] = PR[GP1:90,1] + 59.000;
   1:  PR[GP1:91,2] = PR[GP1:90,2] + 114.505;
   1:L PR[91] 10mm/sec FINE;
   1:  PR[GP1:91,1] = PR[GP1:90,1] + 58.403;
   1:  PR[GP1:91,2] = PR[GP1:90,2] + 112.139;
   1:L PR[91] 10mm/sec FINE;
   1:  PR[GP1:91,1] = PR[GP1:90,1] + 58.205;
   1:  PR[GP1:91,2] = PR[GP1:90,2] + 109.741;
   1:L PR[91] 10mm/sec FINE;
   1:  PR[GP1:91,1] = PR[GP1:90,1] + 58.343;
   1:  PR[GP1:91,2] = PR[GP1:90,2] + 108.907;
   1:L PR[91] 10mm/sec FINE;
   1:  PR[GP1:91,1] = PR[GP1:90,1] + 58.544;
   1:  PR[GP1:91,2] = PR[GP1:90,2] + 106.476;
   1:L PR[91] 10mm/sec FINE;
   1:  PR[GP1:91,1] = PR[GP1:90,1] + 59.135;
   1:  PR[GP1:91,2] = PR[GP1:90,2] + 104.134;
   1:L PR[91] 10mm/sec FINE;
   1:  PR[GP1:91,1] = PR[GP1:90,1] + 60.105;
   1:  PR[GP1:91,2] = PR[GP1:90,2] + 101.914;
   1:L PR[91] 10mm/sec FINE;
   1:  PR[GP1:91,1] = PR[GP1:90,1] + 60.506;
   1:  PR[GP1:91,2] = PR[GP1:90,2] + 101.170;
   1:L PR[91] 10mm/sec FINE;
   1:  PR[GP1:91,1] = PR[GP1:90,1] + 61.827;
   1:  PR[GP1:91,2] = PR[GP1:90,2] + 99.138;
   1:L PR[91] 10mm/sec FINE;
   1:  PR[GP1:91,1] = PR[GP1:90,1] + 63.464;
   1:  PR[GP1:91,2] = PR[GP1:90,2] + 97.351;
   1:L PR[91] 10mm/sec FINE;
   1:  PR[GP1:91,1] = PR[GP1:90,1] + 64.084;
   1:  PR[GP1:91,2] = PR[GP1:90,2] + 96.777;
   1:L PR[91] 10mm/sec FINE;
   1:  PR[GP1:91,1] = PR[GP1:90,1] + 65.991;
   1:  PR[GP1:91,2] = PR[GP1:90,2] + 95.283;
   1:L PR[91] 10mm/sec FINE;
   1:  PR[GP1:91,1] = PR[GP1:90,1] + 68.416;
   1:  PR[GP1:91,2] = PR[GP1:90,2] + 93.959;
   1:  PR[GP1:91,3] = PR[GP1:90,3] + 4.900;
   1:L PR[91] 10mm/sec FINE;
   1:  PR[GP1:91,1] = PR[GP1:90,1] + 68.653;
   1:  PR[GP1:91,2] = PR[GP1:90,2] + 93.858;
   1:L PR[91] 10mm/sec FINE;
   1:  PR[GP1:91,1] = PR[GP1:90,1] + 71.142;
   1:  PR[GP1:91,2] = PR[GP1:90,2] + 92.991;
   1:L PR[91] 10mm/sec FINE;
   1:  PR[GP1:91,1] = PR[GP1:90,1] + 74.009;
   1:  PR[GP1:91,2] = PR[GP1:90,2] + 92.492;
   1:L PR[91] 10mm/sec FINE;
   1:  PR[GP1:91,1] = PR[GP1:90,1] + 76.932;
   1:  PR[GP1:91,2] = PR[GP1:90,2] + 92.484;
   1:L PR[91] 10mm/sec FINE;
   1:  PR[GP1:91,1] = PR[GP1:90,1] + 79.490;
   1:  PR[GP1:91,2] = PR[GP1:90,2] + 92.894;
   1:L PR[91] 10mm/sec FINE;
   1:  PR[GP1:91,1] = PR[GP1:90,1] + 79.822;
   1:  PR[GP1:91,2] = PR[GP1:90,2] + 92.973;
   1:L PR[91] 10mm/sec FINE;
   1:  PR[GP1:91,1] = PR[GP1:90,1] + 82.255;
   1:  PR[GP1:91,2] = PR[GP1:90,2] + 93.791;
   1:L PR[91] 10mm/sec FINE;
   1:  PR[GP1:91,1] = PR[GP1:90,1] + 82.600;
   1:  PR[GP1:91,2] = PR[GP1:90,2] + 93.955;
   1:L PR[91] 10mm/sec FINE;
   1:  PR[GP1:91,1] = PR[GP1:90,1] + 84.844;
   1:  PR[GP1:91,2] = PR[GP1:90,2] + 95.148;
   1:L PR[91] 10mm/sec FINE;
   1:  PR[GP1:91,1] = PR[GP1:90,1] + 87.179;
   1:  PR[GP1:91,2] = PR[GP1:90,2] + 96.938;
   1:L PR[91] 10mm/sec FINE;
   1:  PR[GP1:91,1] = PR[GP1:90,1] + 88.898;
   1:  PR[GP1:91,2] = PR[GP1:90,2] + 98.774;
   1:L PR[91] 10mm/sec FINE;
   1:  PR[GP1:91,1] = PR[GP1:90,1] + 89.178;
   1:  PR[GP1:91,2] = PR[GP1:90,2] + 99.105;
   1:L PR[91] 10mm/sec FINE;
   1:  PR[GP1:91,1] = PR[GP1:90,1] + 90.563;
   1:  PR[GP1:91,2] = PR[GP1:90,2] + 101.183;
   1:L PR[91] 10mm/sec FINE;
   1:  PR[GP1:91,1] = PR[GP1:90,1] + 90.777;
   1:  PR[GP1:91,2] = PR[GP1:90,2] + 101.585;
   1:L PR[91] 10mm/sec FINE;
   1:  PR[GP1:91,1] = PR[GP1:90,1] + 91.798;
   1:  PR[GP1:91,2] = PR[GP1:90,2] + 103.851;
   1:L PR[91] 10mm/sec FINE;
   1:  PR[GP1:91,1] = PR[GP1:90,1] + 92.562;
   1:  PR[GP1:91,2] = PR[GP1:90,2] + 106.735;
   1:L PR[91] 10mm/sec FINE;
   1:  PR[GP1:91,1] = PR[GP1:90,1] + 93.039;
   1:  PR[GP1:91,2] = PR[GP1:90,2] + 107.815;
   1:L PR[91] 10mm/sec FINE;
   1:  PR[GP1:91,1] = PR[GP1:90,1] + 93.094;
   1:  PR[GP1:91,2] = PR[GP1:90,2] + 107.889;
   1:L PR[91] 10mm/sec FINE;
   1:  PR[GP1:91,1] = PR[GP1:90,1] + 94.011;
   1:  PR[GP1:91,2] = PR[GP1:90,2] + 108.652;
   1:L PR[91] 10mm/sec FINE;
   1:  PR[GP1:91,1] = PR[GP1:90,1] + 95.002;
   1:  PR[GP1:91,2] = PR[GP1:90,2] + 108.887;
   1:L PR[91] 10mm/sec FINE;
   1:  PR[GP1:91,1] = PR[GP1:90,1] + 95.102;
   1:  PR[GP1:91,2] = PR[GP1:90,2] + 108.926;
   1:L PR[91] 10mm/sec FINE;
   1:  PR[GP1:91,1] = PR[GP1:90,1] + 95.772;
   1:  PR[GP1:91,2] = PR[GP1:90,2] + 108.932;
   1:L PR[91] 10mm/sec FINE;
   1:  PR[GP1:91,1] = PR[GP1:90,1] + 96.944;
   1:  PR[GP1:91,2] = PR[GP1:90,2] + 108.649;
   1:L PR[91] 10mm/sec FINE;
   1:  PR[GP1:91,1] = PR[GP1:90,1] + 97.903;
   1:  PR[GP1:91,2] = PR[GP1:90,2] + 107.847;
   1:L PR[91] 10mm/sec FINE;
   1:  PR[GP1:91,1] = PR[GP1:90,1] + 98.262;
   1:  PR[GP1:91,2] = PR[GP1:90,2] + 107.015;
   1:L PR[91] 10mm/sec FINE;
   1:  PR[GP1:91,1] = PR[GP1:90,1] + 98.425;
   1:  PR[GP1:91,2] = PR[GP1:90,2] + 106.742;
   1:L PR[91] 10mm/sec FINE;
   1:  PR[GP1:91,1] = PR[GP1:90,1] + 98.629;
   1:  PR[GP1:91,2] = PR[GP1:90,2] + 105.877;
   1:L PR[91] 10mm/sec FINE;
   1:  PR[GP1:91,1] = PR[GP1:90,1] + 99.016;
   1:  PR[GP1:91,2] = PR[GP1:90,2] + 104.405;
   1:L PR[91] 10mm/sec FINE;
   1:  PR[GP1:91,1] = PR[GP1:90,1] + 99.275;
   1:  PR[GP1:91,2] = PR[GP1:90,2] + 103.674;
   1:L PR[91] 10mm/sec FINE;
   1:  PR[GP1:91,1] = PR[GP1:90,1] + 99.864;
   1:  PR[GP1:91,2] = PR[GP1:90,2] + 102.308;
   1:L PR[91] 10mm/sec FINE;
   1:  PR[GP1:91,1] = PR[GP1:90,1] + 100.259;
   1:  PR[GP1:91,2] = PR[GP1:90,2] + 101.493;
   1:L PR[91] 10mm/sec FINE;
   1:  PR[GP1:91,1] = PR[GP1:90,1] + 101.476;
   1:  PR[GP1:91,2] = PR[GP1:90,2] + 99.563;
   1:L PR[91] 10mm/sec FINE;
   1:  PR[GP1:91,1] = PR[GP1:90,1] + 102.134;
   1:  PR[GP1:91,2] = PR[GP1:90,2] + 98.733;
   1:L PR[91] 10mm/sec FINE;
   1:  PR[GP1:91,1] = PR[GP1:90,1] + 102.853;
   1:  PR[GP1:91,2] = PR[GP1:90,2] + 97.911;
   1:L PR[91] 10mm/sec FINE;
   1:  PR[GP1:91,1] = PR[GP1:90,1] + 103.701;
   1:  PR[GP1:91,2] = PR[GP1:90,2] + 97.054;
   1:L PR[91] 10mm/sec FINE;
   1:  PR[GP1:91,1] = PR[GP1:90,1] + 105.388;
   1:  PR[GP1:91,2] = PR[GP1:90,2] + 95.671;
   1:L PR[91] 10mm/sec FINE;
   1:  PR[GP1:91,1] = PR[GP1:90,1] + 106.507;
   1:  PR[GP1:91,2] = PR[GP1:90,2] + 94.953;
   1:L PR[91] 10mm/sec FINE;
   1:  PR[GP1:91,1] = PR[GP1:90,1] + 107.158;
   1:  PR[GP1:91,2] = PR[GP1:90,2] + 94.563;
   1:L PR[91] 10mm/sec FINE;
   1:  PR[GP1:91,1] = PR[GP1:90,1] + 108.435;
   1:  PR[GP1:91,2] = PR[GP1:90,2] + 93.928;
   1:L PR[91] 10mm/sec FINE;
   1:  PR[GP1:91,1] = PR[GP1:90,1] + 108.990;
   1:  PR[GP1:91,2] = PR[GP1:90,2] + 93.705;
   1:L PR[91] 10mm/sec FINE;
   1:  PR[GP1:91,1] = PR[GP1:90,1] + 110.402;
   1:  PR[GP1:91,2] = PR[GP1:90,2] + 93.187;
   1:L PR[91] 10mm/sec FINE;
   1:  PR[GP1:91,1] = PR[GP1:90,1] + 111.864;
   1:  PR[GP1:91,2] = PR[GP1:90,2] + 92.827;
   1:L PR[91] 10mm/sec FINE;
   1:  PR[GP1:91,1] = PR[GP1:90,1] + 112.391;
   1:  PR[GP1:91,2] = PR[GP1:90,2] + 92.706;
   1:L PR[91] 10mm/sec FINE;
   1:  PR[GP1:91,1] = PR[GP1:90,1] + 113.939;
   1:  PR[GP1:91,2] = PR[GP1:90,2] + 92.501;
   1:L PR[91] 10mm/sec FINE;
   1:  PR[GP1:91,1] = PR[GP1:90,1] + 114.380;
   1:  PR[GP1:91,2] = PR[GP1:90,2] + 92.470;
   1:L PR[91] 10mm/sec FINE;
   1:  PR[GP1:91,1] = PR[GP1:90,1] + 115.987;
   1:  PR[GP1:91,2] = PR[GP1:90,2] + 92.434;
   1:L PR[91] 10mm/sec FINE;
   1:  PR[GP1:91,1] = PR[GP1:90,1] + 117.997;
   1:  PR[GP1:91,2] = PR[GP1:90,2] + 92.612;
   1:L PR[91] 10mm/sec FINE;
   1:  PR[GP1:91,1] = PR[GP1:90,1] + 119.608;
   1:  PR[GP1:91,2] = PR[GP1:90,2] + 92.934;
   1:L PR[91] 10mm/sec FINE;
   1:  PR[GP1:91,1] = PR[GP1:90,1] + 119.943;
   1:  PR[GP1:91,2] = PR[GP1:90,2] + 93.017;
   1:L PR[91] 10mm/sec FINE;
   1:  PR[GP1:91,1] = PR[GP1:90,1] + 121.534;
   1:  PR[GP1:91,2] = PR[GP1:90,2] + 93.523;
   1:L PR[91] 10mm/sec FINE;
   1:  PR[GP1:91,1] = PR[GP1:90,1] + 123.361;
   1:  PR[GP1:91,2] = PR[GP1:90,2] + 94.327;
   1:L PR[91] 10mm/sec FINE;
   1:  PR[GP1:91,1] = PR[GP1:90,1] + 124.826;
   1:  PR[GP1:91,2] = PR[GP1:90,2] + 95.180;
   1:L PR[91] 10mm/sec FINE;
   1:  PR[GP1:91,1] = PR[GP1:90,1] + 125.066;
   1:  PR[GP1:91,2] = PR[GP1:90,2] + 95.329;
   1:L PR[91] 10mm/sec FINE;
   1:  PR[GP1:91,1] = PR[GP1:90,1] + 126.441;
   1:  PR[GP1:91,2] = PR[GP1:90,2] + 96.347;
   1:L PR[91] 10mm/sec FINE;
   1:  PR[GP1:91,1] = PR[GP1:90,1] + 126.633;
   1:  PR[GP1:91,2] = PR[GP1:90,2] + 96.513;
   1:L PR[91] 10mm/sec FINE;
   1:  PR[GP1:91,1] = PR[GP1:90,1] + 127.899;
   1:  PR[GP1:91,2] = PR[GP1:90,2] + 97.685;
   1:L PR[91] 10mm/sec FINE;
   1:  PR[GP1:91,1] = PR[GP1:90,1] + 129.189;
   1:  PR[GP1:91,2] = PR[GP1:90,2] + 99.178;
   1:L PR[91] 10mm/sec FINE;
   1:  PR[GP1:91,1] = PR[GP1:90,1] + 130.174;
   1:  PR[GP1:91,2] = PR[GP1:90,2] + 100.605;
   1:L PR[91] 10mm/sec FINE;
   1:  PR[GP1:91,1] = PR[GP1:90,1] + 130.291;
   1:  PR[GP1:91,2] = PR[GP1:90,2] + 100.798;
   1:L PR[91] 10mm/sec FINE;
   1:  PR[GP1:91,1] = PR[GP1:90,1] + 131.118;
   1:  PR[GP1:91,2] = PR[GP1:90,2] + 102.332;
   1:L PR[91] 10mm/sec FINE;
   1:  PR[GP1:91,1] = PR[GP1:90,1] + 131.856;
   1:  PR[GP1:91,2] = PR[GP1:90,2] + 104.154;
   1:L PR[91] 10mm/sec FINE;
   1:  PR[GP1:91,1] = PR[GP1:90,1] + 132.380;
   1:  PR[GP1:91,2] = PR[GP1:90,2] + 106.046;
   1:L PR[91] 10mm/sec FINE;
   1:  PR[GP1:91,1] = PR[GP1:90,1] + 132.666;
   1:  PR[GP1:91,2] = PR[GP1:90,2] + 107.770;
   1:L PR[91] 10mm/sec FINE;
   1:  PR[GP1:91,1] = PR[GP1:90,1] + 132.783;
   1:  PR[GP1:91,2] = PR[GP1:90,2] + 109.726;
   1:L PR[91] 10mm/sec FINE;
   1:  PR[GP1:91,1] = PR[GP1:90,1] + 132.442;
   1:  PR[GP1:91,2] = PR[GP1:90,2] + 113.131;
   1:L PR[91] 10mm/sec FINE;
   1:  PR[GP1:91,1] = PR[GP1:90,1] + 131.814;
   1:  PR[GP1:91,2] = PR[GP1:90,2] + 115.422;
   1:L PR[91] 10mm/sec FINE;
   1:  PR[GP1:91,1] = PR[GP1:90,1] + 131.446;
   1:  PR[GP1:91,2] = PR[GP1:90,2] + 116.391;
   1:L PR[91] 10mm/sec FINE;
   1:  PR[GP1:91,1] = PR[GP1:90,1] + 129.820;
   1:  PR[GP1:91,2] = PR[GP1:90,2] + 119.406;
   1:L PR[91] 10mm/sec FINE;
   1:  PR[GP1:91,1] = PR[GP1:90,1] + 129.626;
   1:  PR[GP1:91,2] = PR[GP1:90,2] + 119.639;
   1:L PR[91] 10mm/sec FINE;
   1:  PR[GP1:91,1] = PR[GP1:90,1] + 129.018;
   1:  PR[GP1:91,2] = PR[GP1:90,2] + 120.480;
   1:L PR[91] 10mm/sec FINE;
   1:  PR[GP1:91,1] = PR[GP1:90,1] + 127.640;
   1:  PR[GP1:91,2] = PR[GP1:90,2] + 122.034;
   1:L PR[91] 10mm/sec FINE;
   1:  PR[GP1:91,1] = PR[GP1:90,1] + 124.980;
   1:  PR[GP1:91,2] = PR[GP1:90,2] + 124.187;
   1:L PR[91] 10mm/sec FINE;
   1:  PR[GP1:91,1] = PR[GP1:90,1] + 121.952;
   1:  PR[GP1:91,2] = PR[GP1:90,2] + 125.773;
   1:L PR[91] 10mm/sec FINE;
   1:  PR[GP1:91,1] = PR[GP1:90,1] + 121.559;
   1:  PR[GP1:91,2] = PR[GP1:90,2] + 125.888;
   1:L PR[91] 10mm/sec FINE;
   1:  PR[GP1:91,1] = PR[GP1:90,1] + 119.661;
   1:  PR[GP1:91,2] = PR[GP1:90,2] + 126.513;
   1:L PR[91] 10mm/sec FINE;
   1:  PR[GP1:91,1] = PR[GP1:90,1] + 118.679;
   1:  PR[GP1:91,2] = PR[GP1:90,2] + 126.731;
   1:L PR[91] 10mm/sec FINE;
   1:  PR[GP1:91,1] = PR[GP1:90,1] + 115.266;
   1:  PR[GP1:91,2] = PR[GP1:90,2] + 127.028;
   1:L PR[91] 10mm/sec FINE;
   1:  PR[GP1:91,1] = PR[GP1:90,1] + 114.719;
   1:  PR[GP1:91,2] = PR[GP1:90,2] + 126.966;
   1:L PR[91] 10mm/sec FINE;
   1:  PR[GP1:91,1] = PR[GP1:90,1] + 113.778;
   1:  PR[GP1:91,2] = PR[GP1:90,2] + 126.925;
   1:L PR[91] 10mm/sec FINE;
   1:  PR[GP1:91,1] = PR[GP1:90,1] + 111.873;
   1:  PR[GP1:91,2] = PR[GP1:90,2] + 126.649;
   1:L PR[91] 10mm/sec FINE;
   1:  PR[GP1:91,1] = PR[GP1:90,1] + 108.637;
   1:  PR[GP1:91,2] = PR[GP1:90,2] + 125.618;
   1:L PR[91] 10mm/sec FINE;
   1:  PR[GP1:91,1] = PR[GP1:90,1] + 105.627;
   1:  PR[GP1:91,2] = PR[GP1:90,2] + 123.948;
   1:L PR[91] 10mm/sec FINE;
   1:  PR[GP1:91,1] = PR[GP1:90,1] + 104.806;
   1:  PR[GP1:91,2] = PR[GP1:90,2] + 123.250;
   1:L PR[91] 10mm/sec FINE;
   1:  PR[GP1:91,1] = PR[GP1:90,1] + 103.596;
   1:  PR[GP1:91,2] = PR[GP1:90,2] + 122.289;
   1:L PR[91] 10mm/sec FINE;
   1:  PR[GP1:91,1] = PR[GP1:90,1] + 103.028;
   1:  PR[GP1:91,2] = PR[GP1:90,2] + 121.739;
   1:L PR[91] 10mm/sec FINE;
   1:  PR[GP1:91,1] = PR[GP1:90,1] + 100.906;
   1:  PR[GP1:91,2] = PR[GP1:90,2] + 119.050;
   1:L PR[91] 10mm/sec FINE;
   1:  PR[GP1:91,1] = PR[GP1:90,1] + 100.087;
   1:  PR[GP1:91,2] = PR[GP1:90,2] + 117.438;
   1:L PR[91] 10mm/sec FINE;
   1:  PR[GP1:91,1] = PR[GP1:90,1] + 99.820;
   1:  PR[GP1:91,2] = PR[GP1:90,2] + 116.989;
   1:L PR[91] 10mm/sec FINE;
   1:  PR[GP1:91,1] = PR[GP1:90,1] + 99.359;
   1:  PR[GP1:91,2] = PR[GP1:90,2] + 116.006;
   1:L PR[91] 10mm/sec FINE;
   1:  PR[GP1:91,1] = PR[GP1:90,1] + 98.437;
   1:  PR[GP1:91,2] = PR[GP1:90,2] + 112.726;
   1:L PR[91] 10mm/sec FINE;
   1:  PR[GP1:91,1] = PR[GP1:90,1] + 98.256;
   1:  PR[GP1:91,2] = PR[GP1:90,2] + 112.308;
   1:L PR[91] 10mm/sec FINE;
   1:  PR[GP1:91,1] = PR[GP1:90,1] + 98.026;
   1:  PR[GP1:91,2] = PR[GP1:90,2] + 111.873;
   1:L PR[91] 10mm/sec FINE;
   1:  PR[GP1:91,1] = PR[GP1:90,1] + 97.909;
   1:  PR[GP1:91,2] = PR[GP1:90,2] + 111.611;
   1:L PR[91] 10mm/sec FINE;
   1:  PR[GP1:91,1] = PR[GP1:90,1] + 96.953;
   1:  PR[GP1:91,2] = PR[GP1:90,2] + 110.813;
   1:L PR[91] 10mm/sec FINE;
   1:  PR[GP1:91,1] = PR[GP1:90,1] + 95.781;
   1:  PR[GP1:91,2] = PR[GP1:90,2] + 110.532;
   1:L PR[91] 10mm/sec FINE;
   1:  PR[GP1:91,1] = PR[GP1:90,1] + 95.180;
   1:L PR[91] 10mm/sec FINE;
   1:  PR[GP1:91,1] = PR[GP1:90,1] + 94.154;
   1:  PR[GP1:91,2] = PR[GP1:90,2] + 110.767;
   1:L PR[91] 10mm/sec FINE;
   1:  PR[GP1:91,1] = PR[GP1:90,1] + 93.983;
   1:  PR[GP1:91,2] = PR[GP1:90,2] + 110.828;
   1:L PR[91] 10mm/sec FINE;
   1:  PR[GP1:91,1] = PR[GP1:90,1] + 93.138;
   1:  PR[GP1:91,2] = PR[GP1:90,2] + 111.532;
   1:L PR[91] 10mm/sec FINE;
   1:  PR[GP1:91,1] = PR[GP1:90,1] + 93.043;
   1:  PR[GP1:91,2] = PR[GP1:90,2] + 111.634;
   1:L PR[91] 10mm/sec FINE;
   1:  PR[GP1:91,1] = PR[GP1:90,1] + 92.628;
   1:  PR[GP1:91,2] = PR[GP1:90,2] + 112.600;
   1:L PR[91] 10mm/sec FINE;
   1:  PR[GP1:91,1] = PR[GP1:90,1] + 92.592;
   1:  PR[GP1:91,2] = PR[GP1:90,2] + 112.602;
   1:L PR[91] 10mm/sec FINE;
   1:  PR[GP1:91,1] = PR[GP1:90,1] + 91.916;
   1:  PR[GP1:91,2] = PR[GP1:90,2] + 115.190;
   1:L PR[91] 10mm/sec FINE;
   1:  PR[GP1:91,1] = PR[GP1:90,1] + 91.799;
   1:  PR[GP1:91,2] = PR[GP1:90,2] + 115.594;
   1:L PR[91] 10mm/sec FINE;
   1:  PR[GP1:91,1] = PR[GP1:90,1] + 90.758;
   1:  PR[GP1:91,2] = PR[GP1:90,2] + 117.907;
   1:L PR[91] 10mm/sec FINE;
   1:  PR[GP1:91,1] = PR[GP1:90,1] + 90.577;
   1:  PR[GP1:91,2] = PR[GP1:90,2] + 118.243;
   1:L PR[91] 10mm/sec FINE;
   1:  PR[GP1:91,1] = PR[GP1:90,1] + 89.155;
   1:  PR[GP1:91,2] = PR[GP1:90,2] + 120.376;
   1:L PR[91] 10mm/sec FINE;
   1:  PR[GP1:91,1] = PR[GP1:90,1] + 88.935;
   1:  PR[GP1:91,2] = PR[GP1:90,2] + 120.635;
   1:L PR[91] 10mm/sec FINE;
   1:  PR[GP1:91,1] = PR[GP1:90,1] + 87.164;
   1:  PR[GP1:91,2] = PR[GP1:90,2] + 122.525;
   1:L PR[91] 10mm/sec FINE;
   1:  PR[GP1:91,1] = PR[GP1:90,1] + 84.846;
   1:  PR[GP1:91,2] = PR[GP1:90,2] + 124.300;
   1:L PR[91] 10mm/sec FINE;
   1:  PR[GP1:91,1] = PR[GP1:90,1] + 82.538;
   1:  PR[GP1:91,2] = PR[GP1:90,2] + 125.527;
   1:L PR[91] 10mm/sec FINE;
   1:  PR[GP1:91,1] = PR[GP1:90,1] + 82.277;
   1:  PR[GP1:91,2] = PR[GP1:90,2] + 125.650;
   1:L PR[91] 10mm/sec FINE;
   1:  PR[GP1:91,1] = PR[GP1:90,1] + 79.779;
   1:  PR[GP1:91,2] = PR[GP1:90,2] + 126.489;
   1:L PR[91] 10mm/sec FINE;
   1:  PR[GP1:91,1] = PR[GP1:90,1] + 79.528;
   1:  PR[GP1:91,2] = PR[GP1:90,2] + 126.548;
   1:L PR[91] 10mm/sec FINE;
   1:  PR[GP1:91,1] = PR[GP1:90,1] + 76.910;
   1:  PR[GP1:91,2] = PR[GP1:90,2] + 126.968;
   1:L PR[91] 10mm/sec FINE;
   1:  PR[GP1:91,1] = PR[GP1:90,1] + 74.005;
   1:  PR[GP1:91,2] = PR[GP1:90,2] + 126.958;
   1:L PR[91] 10mm/sec FINE;
   1:  PR[GP1:91,1] = PR[GP1:90,1] + 71.151;
   1:  PR[GP1:91,2] = PR[GP1:90,2] + 126.461;
   1:L PR[91] 10mm/sec FINE;
   1:  PR[GP1:91,1] = PR[GP1:90,1] + 68.622;
   1:  PR[GP1:91,2] = PR[GP1:90,2] + 125.580;
   1:L PR[91] 10mm/sec FINE;
   1:  PR[GP1:91,1] = PR[GP1:90,1] + 68.431;
   1:  PR[GP1:91,2] = PR[GP1:90,2] + 125.498;
   1:L PR[91] 10mm/sec FINE;
   1:  PR[GP1:91,1] = PR[GP1:90,1] + 66.075;
   1:  PR[GP1:91,2] = PR[GP1:90,2] + 124.211;
   1:L PR[91] 10mm/sec FINE;
   1:  PR[GP1:91,1] = PR[GP1:90,1] + 63.789;
   1:  PR[GP1:91,2] = PR[GP1:90,2] + 122.433;
   1:L PR[91] 10mm/sec FINE;
   1:  PR[GP1:91,1] = PR[GP1:90,1] + 61.836;
   1:  PR[GP1:91,2] = PR[GP1:90,2] + 120.300;
   1:L PR[91] 10mm/sec FINE;
   1:  PR[GP1:91,1] = PR[GP1:90,1] + 60.268;
   1:  PR[GP1:91,2] = PR[GP1:90,2] + 117.871;
   1:L PR[91] 10mm/sec FINE;
   1:  PR[GP1:91,1] = PR[GP1:90,1] + 59.188;
   1:  PR[GP1:91,2] = PR[GP1:90,2] + 115.399;
   1:L PR[91] 10mm/sec FINE;
   1:  PR[GP1:91,1] = PR[GP1:90,1] + 59.130;
   1:  PR[GP1:91,2] = PR[GP1:90,2] + 115.224;
   1:L PR[91] 10mm/sec FINE;
   1:  PR[GP1:91,1] = PR[GP1:90,1] + 58.470;
   1:  PR[GP1:91,2] = PR[GP1:90,2] + 112.606;
   1:L PR[91] 10mm/sec FINE;
   1:  PR[GP1:91,1] = PR[GP1:90,1] + 58.227;
   1:  PR[GP1:91,2] = PR[GP1:90,2] + 109.725;
   1:L PR[91] 10mm/sec FINE;
   1:  PR[GP1:91,1] = PR[GP1:90,1] + 58.470;
   1:  PR[GP1:91,2] = PR[GP1:90,2] + 106.841;
   1:L PR[91] 10mm/sec FINE;
   1:  PR[GP1:91,1] = PR[GP1:90,1] + 59.129;
   1:  PR[GP1:91,2] = PR[GP1:90,2] + 104.230;
   1:L PR[91] 10mm/sec FINE;
   1:  PR[GP1:91,1] = PR[GP1:90,1] + 59.191;
   1:  PR[GP1:91,2] = PR[GP1:90,2] + 104.043;
   1:L PR[91] 10mm/sec FINE;
   1:  PR[GP1:91,1] = PR[GP1:90,1] + 60.268;
   1:  PR[GP1:91,2] = PR[GP1:90,2] + 101.578;
   1:L PR[91] 10mm/sec FINE;
   1:  PR[GP1:91,1] = PR[GP1:90,1] + 60.373;
   1:  PR[GP1:91,2] = PR[GP1:90,2] + 101.399;
   1:L PR[91] 10mm/sec FINE;
   1:  PR[GP1:91,1] = PR[GP1:90,1] + 61.835;
   1:  PR[GP1:91,2] = PR[GP1:90,2] + 99.151;
   1:L PR[91] 10mm/sec FINE;
   1:  PR[GP1:91,1] = PR[GP1:90,1] + 63.794;
   1:  PR[GP1:91,2] = PR[GP1:90,2] + 97.013;
   1:L PR[91] 10mm/sec FINE;
   1:  PR[GP1:91,1] = PR[GP1:90,1] + 65.895;
   1:  PR[GP1:91,2] = PR[GP1:90,2] + 95.366;
   1:L PR[91] 10mm/sec FINE;
   1:  PR[GP1:91,1] = PR[GP1:90,1] + 66.085;
   1:  PR[GP1:91,2] = PR[GP1:90,2] + 95.232;
   1:L PR[91] 10mm/sec FINE;
   1:  PR[GP1:91,1] = PR[GP1:90,1] + 68.216;
   1:  PR[GP1:91,2] = PR[GP1:90,2] + 94.069;
   1:  PR[GP1:91,3] = PR[GP1:90,3] + 5.900;
   1:L PR[91] 10mm/sec FINE;
   1:  PR[GP1:91,1] = PR[GP1:90,1] + 69.085;
   1:  PR[GP1:91,2] = PR[GP1:90,2] + 93.699;
   1:L PR[91] 10mm/sec FINE;
   1:  PR[GP1:91,1] = PR[GP1:90,1] + 71.053;
   1:  PR[GP1:91,2] = PR[GP1:90,2] + 93.014;
   1:L PR[91] 10mm/sec FINE;
   1:  PR[GP1:91,1] = PR[GP1:90,1] + 73.115;
   1:  PR[GP1:91,2] = PR[GP1:90,2] + 92.659;
   1:L PR[91] 10mm/sec FINE;
   1:  PR[GP1:91,1] = PR[GP1:90,1] + 74.076;
   1:  PR[GP1:91,2] = PR[GP1:90,2] + 92.471;
   1:L PR[91] 10mm/sec FINE;
   1:  PR[GP1:91,1] = PR[GP1:90,1] + 76.088;
   1:  PR[GP1:91,2] = PR[GP1:90,2] + 92.460;
   1:L PR[91] 10mm/sec FINE;
   1:  PR[GP1:91,1] = PR[GP1:90,1] + 77.185;
   1:  PR[GP1:91,2] = PR[GP1:90,2] + 92.483;
   1:L PR[91] 10mm/sec FINE;
   1:  PR[GP1:91,1] = PR[GP1:90,1] + 79.090;
   1:  PR[GP1:91,2] = PR[GP1:90,2] + 92.789;
   1:L PR[91] 10mm/sec FINE;
   1:  PR[GP1:91,1] = PR[GP1:90,1] + 80.289;
   1:  PR[GP1:91,2] = PR[GP1:90,2] + 93.075;
   1:L PR[91] 10mm/sec FINE;
   1:  PR[GP1:91,1] = PR[GP1:90,1] + 82.032;
   1:  PR[GP1:91,2] = PR[GP1:90,2] + 93.660;
   1:L PR[91] 10mm/sec FINE;
   1:  PR[GP1:91,1] = PR[GP1:90,1] + 83.276;
   1:  PR[GP1:91,2] = PR[GP1:90,2] + 94.254;
   1:L PR[91] 10mm/sec FINE;
   1:  PR[GP1:91,1] = PR[GP1:90,1] + 84.816;
   1:  PR[GP1:91,2] = PR[GP1:90,2] + 95.073;
   1:L PR[91] 10mm/sec FINE;
   1:  PR[GP1:91,1] = PR[GP1:90,1] + 87.339;
   1:  PR[GP1:91,2] = PR[GP1:90,2] + 97.009;
   1:L PR[91] 10mm/sec FINE;
   1:  PR[GP1:91,1] = PR[GP1:90,1] + 88.473;
   1:  PR[GP1:91,2] = PR[GP1:90,2] + 98.220;
   1:L PR[91] 10mm/sec FINE;
   1:  PR[GP1:91,1] = PR[GP1:90,1] + 89.477;
   1:  PR[GP1:91,2] = PR[GP1:90,2] + 99.409;
   1:L PR[91] 10mm/sec FINE;
   1:  PR[GP1:91,1] = PR[GP1:90,1] + 90.361;
   1:  PR[GP1:91,2] = PR[GP1:90,2] + 100.735;
   1:L PR[91] 10mm/sec FINE;
   1:  PR[GP1:91,1] = PR[GP1:90,1] + 91.132;
   1:  PR[GP1:91,2] = PR[GP1:90,2] + 102.179;
   1:L PR[91] 10mm/sec FINE;
   1:  PR[GP1:91,1] = PR[GP1:90,1] + 91.771;
   1:  PR[GP1:91,2] = PR[GP1:90,2] + 103.598;
   1:L PR[91] 10mm/sec FINE;
   1:  PR[GP1:91,1] = PR[GP1:90,1] + 92.612;
   1:  PR[GP1:91,2] = PR[GP1:90,2] + 106.754;
   1:L PR[91] 10mm/sec FINE;
   1:  PR[GP1:91,1] = PR[GP1:90,1] + 92.700;
   1:  PR[GP1:91,2] = PR[GP1:90,2] + 106.876;
   1:L PR[91] 10mm/sec FINE;
   1:  PR[GP1:91,1] = PR[GP1:90,1] + 93.094;
   1:  PR[GP1:91,2] = PR[GP1:90,2] + 107.781;
   1:L PR[91] 10mm/sec FINE;
   1:  PR[GP1:91,1] = PR[GP1:90,1] + 93.219;
   1:  PR[GP1:91,2] = PR[GP1:90,2] + 107.949;
   1:L PR[91] 10mm/sec FINE;
   1:  PR[GP1:91,1] = PR[GP1:90,1] + 93.745;
   1:  PR[GP1:91,2] = PR[GP1:90,2] + 108.390;
   1:L PR[91] 10mm/sec FINE;
   1:  PR[GP1:91,1] = PR[GP1:90,1] + 93.822;
   1:  PR[GP1:91,2] = PR[GP1:90,2] + 108.473;
   1:L PR[91] 10mm/sec FINE;
   1:  PR[GP1:91,1] = PR[GP1:90,1] + 94.092;
   1:  PR[GP1:91,2] = PR[GP1:90,2] + 108.659;
   1:L PR[91] 10mm/sec FINE;
   1:  PR[GP1:91,1] = PR[GP1:90,1] + 94.656;
   1:  PR[GP1:91,2] = PR[GP1:90,2] + 108.793;
   1:L PR[91] 10mm/sec FINE;
   1:  PR[GP1:91,1] = PR[GP1:90,1] + 94.766;
   1:  PR[GP1:91,2] = PR[GP1:90,2] + 108.850;
   1:L PR[91] 10mm/sec FINE;
   1:  PR[GP1:91,1] = PR[GP1:90,1] + 94.972;
   1:  PR[GP1:91,2] = PR[GP1:90,2] + 108.910;
   1:L PR[91] 10mm/sec FINE;
   1:  PR[GP1:91,1] = PR[GP1:90,1] + 95.447;
   1:  PR[GP1:91,2] = PR[GP1:90,2] + 108.933;
   1:L PR[91] 10mm/sec FINE;
   1:  PR[GP1:91,1] = PR[GP1:90,1] + 96.742;
   1:  PR[GP1:91,2] = PR[GP1:90,2] + 108.641;
   1:L PR[91] 10mm/sec FINE;
   1:  PR[GP1:91,1] = PR[GP1:90,1] + 97.705;
   1:  PR[GP1:91,2] = PR[GP1:90,2] + 107.841;
   1:L PR[91] 10mm/sec FINE;
   1:  PR[GP1:91,1] = PR[GP1:90,1] + 98.233;
   1:  PR[GP1:91,2] = PR[GP1:90,2] + 106.719;
   1:L PR[91] 10mm/sec FINE;
   1:  PR[GP1:91,1] = PR[GP1:90,1] + 98.925;
   1:  PR[GP1:91,2] = PR[GP1:90,2] + 104.071;
   1:L PR[91] 10mm/sec FINE;
   1:  PR[GP1:91,1] = PR[GP1:90,1] + 100.017;
   1:  PR[GP1:91,2] = PR[GP1:90,2] + 101.591;
   1:L PR[91] 10mm/sec FINE;
   1:  PR[GP1:91,1] = PR[GP1:90,1] + 101.490;
   1:  PR[GP1:91,2] = PR[GP1:90,2] + 99.313;
   1:L PR[91] 10mm/sec FINE;
   1:  PR[GP1:91,1] = PR[GP1:90,1] + 103.306;
   1:  PR[GP1:91,2] = PR[GP1:90,2] + 97.291;
   1:L PR[91] 10mm/sec FINE;
   1:  PR[GP1:91,1] = PR[GP1:90,1] + 105.420;
   1:  PR[GP1:91,2] = PR[GP1:90,2] + 95.574;
   1:L PR[91] 10mm/sec FINE;
   1:  PR[GP1:91,1] = PR[GP1:90,1] + 107.647;
   1:  PR[GP1:91,2] = PR[GP1:90,2] + 94.252;
   1:L PR[91] 10mm/sec FINE;
   1:  PR[GP1:91,1] = PR[GP1:90,1] + 107.850;
   1:  PR[GP1:91,2] = PR[GP1:90,2] + 94.150;
   1:L PR[91] 10mm/sec FINE;
   1:  PR[GP1:91,1] = PR[GP1:90,1] + 109.820;
   1:  PR[GP1:91,2] = PR[GP1:90,2] + 93.357;
   1:L PR[91] 10mm/sec FINE;
   1:  PR[GP1:91,1] = PR[GP1:90,1] + 110.286;
   1:  PR[GP1:91,2] = PR[GP1:90,2] + 93.186;
   1:L PR[91] 10mm/sec FINE;
   1:  PR[GP1:91,1] = PR[GP1:90,1] + 110.768;
   1:  PR[GP1:91,2] = PR[GP1:90,2] + 93.068;
   1:L PR[91] 10mm/sec FINE;
   1:  PR[GP1:91,1] = PR[GP1:90,1] + 112.640;
   1:  PR[GP1:91,2] = PR[GP1:90,2] + 92.637;
   1:L PR[91] 10mm/sec FINE;
   1:  PR[GP1:91,1] = PR[GP1:90,1] + 113.335;
   1:  PR[GP1:91,2] = PR[GP1:90,2] + 92.545;
   1:L PR[91] 10mm/sec FINE;
   1:  PR[GP1:91,1] = PR[GP1:90,1] + 114.907;
   1:  PR[GP1:91,2] = PR[GP1:90,2] + 92.435;
   1:L PR[91] 10mm/sec FINE;
   1:  PR[GP1:91,1] = PR[GP1:90,1] + 115.768;
   1:  PR[GP1:91,2] = PR[GP1:90,2] + 92.416;
   1:L PR[91] 10mm/sec FINE;
   1:  PR[GP1:91,1] = PR[GP1:90,1] + 118.073;
   1:  PR[GP1:91,2] = PR[GP1:90,2] + 92.618;
   1:L PR[91] 10mm/sec FINE;
   1:  PR[GP1:91,1] = PR[GP1:90,1] + 119.040;
   1:  PR[GP1:91,2] = PR[GP1:90,2] + 92.812;
   1:L PR[91] 10mm/sec FINE;
   1:  PR[GP1:91,1] = PR[GP1:90,1] + 120.238;
   1:  PR[GP1:91,2] = PR[GP1:90,2] + 93.109;
   1:L PR[91] 10mm/sec FINE;
   1:  PR[GP1:91,1] = PR[GP1:90,1] + 121.271;
   1:  PR[GP1:91,2] = PR[GP1:90,2] + 93.437;
   1:L PR[91] 10mm/sec FINE;
   1:  PR[GP1:91,1] = PR[GP1:90,1] + 123.328;
   1:  PR[GP1:91,2] = PR[GP1:90,2] + 94.328;
   1:L PR[91] 10mm/sec FINE;
   1:  PR[GP1:91,1] = PR[GP1:90,1] + 124.333;
   1:  PR[GP1:91,2] = PR[GP1:90,2] + 94.914;
   1:L PR[91] 10mm/sec FINE;
   1:  PR[GP1:91,1] = PR[GP1:90,1] + 125.197;
   1:  PR[GP1:91,2] = PR[GP1:90,2] + 95.450;
   1:L PR[91] 10mm/sec FINE;
   1:  PR[GP1:91,1] = PR[GP1:90,1] + 126.180;
   1:  PR[GP1:91,2] = PR[GP1:90,2] + 96.178;
   1:L PR[91] 10mm/sec FINE;
   1:  PR[GP1:91,1] = PR[GP1:90,1] + 126.873;
   1:  PR[GP1:91,2] = PR[GP1:90,2] + 96.776;
   1:L PR[91] 10mm/sec FINE;
   1:  PR[GP1:91,1] = PR[GP1:90,1] + 127.807;
   1:  PR[GP1:91,2] = PR[GP1:90,2] + 97.641;
   1:L PR[91] 10mm/sec FINE;
   1:  PR[GP1:91,1] = PR[GP1:90,1] + 129.210;
   1:  PR[GP1:91,2] = PR[GP1:90,2] + 99.276;
   1:L PR[91] 10mm/sec FINE;
   1:  PR[GP1:91,1] = PR[GP1:90,1] + 129.954;
   1:  PR[GP1:91,2] = PR[GP1:90,2] + 100.353;
   1:L PR[91] 10mm/sec FINE;
   1:  PR[GP1:91,1] = PR[GP1:90,1] + 130.377;
   1:  PR[GP1:91,2] = PR[GP1:90,2] + 101.051;
   1:L PR[91] 10mm/sec FINE;
   1:  PR[GP1:91,1] = PR[GP1:90,1] + 131.012;
   1:  PR[GP1:91,2] = PR[GP1:90,2] + 102.228;
   1:L PR[91] 10mm/sec FINE;
   1:  PR[GP1:91,1] = PR[GP1:90,1] + 131.816;
   1:  PR[GP1:91,2] = PR[GP1:90,2] + 104.206;
   1:L PR[91] 10mm/sec FINE;
   1:  PR[GP1:91,1] = PR[GP1:90,1] + 132.185;
   1:  PR[GP1:91,2] = PR[GP1:90,2] + 105.515;
   1:L PR[91] 10mm/sec FINE;
   1:  PR[GP1:91,1] = PR[GP1:90,1] + 132.360;
   1:  PR[GP1:91,2] = PR[GP1:90,2] + 106.252;
   1:L PR[91] 10mm/sec FINE;
   1:  PR[GP1:91,1] = PR[GP1:90,1] + 132.585;
   1:  PR[GP1:91,2] = PR[GP1:90,2] + 107.605;
   1:L PR[91] 10mm/sec FINE;
   1:  PR[GP1:91,1] = PR[GP1:90,1] + 132.661;
   1:  PR[GP1:91,2] = PR[GP1:90,2] + 108.985;
   1:L PR[91] 10mm/sec FINE;
   1:  PR[GP1:91,1] = PR[GP1:90,1] + 132.733;
   1:  PR[GP1:91,2] = PR[GP1:90,2] + 109.725;
   1:L PR[91] 10mm/sec FINE;
   1:  PR[GP1:91,1] = PR[GP1:90,1] + 132.385;
   1:  PR[GP1:91,2] = PR[GP1:90,2] + 113.123;
   1:L PR[91] 10mm/sec FINE;
   1:  PR[GP1:91,1] = PR[GP1:90,1] + 132.091;
   1:  PR[GP1:91,2] = PR[GP1:90,2] + 114.082;
   1:L PR[91] 10mm/sec FINE;
   1:  PR[GP1:91,1] = PR[GP1:90,1] + 131.669;
   1:  PR[GP1:91,2] = PR[GP1:90,2] + 115.645;
   1:L PR[91] 10mm/sec FINE;
   1:  PR[GP1:91,1] = PR[GP1:90,1] + 131.388;
   1:  PR[GP1:91,2] = PR[GP1:90,2] + 116.387;
   1:L PR[91] 10mm/sec FINE;
   1:  PR[GP1:91,1] = PR[GP1:90,1] + 129.761;
   1:  PR[GP1:91,2] = PR[GP1:90,2] + 119.401;
   1:L PR[91] 10mm/sec FINE;
   1:  PR[GP1:91,1] = PR[GP1:90,1] + 129.062;
   1:  PR[GP1:91,2] = PR[GP1:90,2] + 120.242;
   1:L PR[91] 10mm/sec FINE;
   1:  PR[GP1:91,1] = PR[GP1:90,1] + 128.607;
   1:  PR[GP1:91,2] = PR[GP1:90,2] + 120.871;
   1:L PR[91] 10mm/sec FINE;
   1:  PR[GP1:91,1] = PR[GP1:90,1] + 127.580;
   1:  PR[GP1:91,2] = PR[GP1:90,2] + 122.030;
   1:L PR[91] 10mm/sec FINE;
   1:  PR[GP1:91,1] = PR[GP1:90,1] + 124.920;
   1:  PR[GP1:91,2] = PR[GP1:90,2] + 124.182;
   1:L PR[91] 10mm/sec FINE;
   1:  PR[GP1:91,1] = PR[GP1:90,1] + 121.893;
   1:  PR[GP1:91,2] = PR[GP1:90,2] + 125.768;
   1:L PR[91] 10mm/sec FINE;
   1:  PR[GP1:91,1] = PR[GP1:90,1] + 120.475;
   1:  PR[GP1:91,2] = PR[GP1:90,2] + 126.183;
   1:L PR[91] 10mm/sec FINE;
   1:  PR[GP1:91,1] = PR[GP1:90,1] + 119.248;
   1:  PR[GP1:91,2] = PR[GP1:90,2] + 126.587;
   1:L PR[91] 10mm/sec FINE;
   1:  PR[GP1:91,1] = PR[GP1:90,1] + 118.620;
   1:  PR[GP1:91,2] = PR[GP1:90,2] + 126.726;
   1:L PR[91] 10mm/sec FINE;
   1:  PR[GP1:91,1] = PR[GP1:90,1] + 115.204;
   1:  PR[GP1:91,2] = PR[GP1:90,2] + 127.022;
   1:L PR[91] 10mm/sec FINE;
   1:  PR[GP1:91,1] = PR[GP1:90,1] + 113.256;
   1:  PR[GP1:91,2] = PR[GP1:90,2] + 126.804;
   1:L PR[91] 10mm/sec FINE;
   1:  PR[GP1:91,1] = PR[GP1:90,1] + 112.776;
   1:  PR[GP1:91,2] = PR[GP1:90,2] + 126.783;
   1:L PR[91] 10mm/sec FINE;
   1:  PR[GP1:91,1] = PR[GP1:90,1] + 111.814;
   1:  PR[GP1:91,2] = PR[GP1:90,2] + 126.644;
   1:L PR[91] 10mm/sec FINE;
   1:  PR[GP1:91,1] = PR[GP1:90,1] + 108.553;
   1:  PR[GP1:91,2] = PR[GP1:90,2] + 125.603;
   1:L PR[91] 10mm/sec FINE;
   1:  PR[GP1:91,1] = PR[GP1:90,1] + 105.569;
   1:  PR[GP1:91,2] = PR[GP1:90,2] + 123.943;
   1:L PR[91] 10mm/sec FINE;
   1:  PR[GP1:91,1] = PR[GP1:90,1] + 102.950;
   1:  PR[GP1:91,2] = PR[GP1:90,2] + 121.726;
   1:L PR[91] 10mm/sec FINE;
   1:  PR[GP1:91,1] = PR[GP1:90,1] + 100.799;
   1:  PR[GP1:91,2] = PR[GP1:90,2] + 119.039;
   1:L PR[91] 10mm/sec FINE;
   1:  PR[GP1:91,1] = PR[GP1:90,1] + 99.222;
   1:  PR[GP1:91,2] = PR[GP1:90,2] + 115.988;
   1:L PR[91] 10mm/sec FINE;
   1:  PR[GP1:91,1] = PR[GP1:90,1] + 98.265;
   1:  PR[GP1:91,2] = PR[GP1:90,2] + 112.701;
   1:L PR[91] 10mm/sec FINE;
   1:  PR[GP1:91,1] = PR[GP1:90,1] + 98.098;
   1:  PR[GP1:91,2] = PR[GP1:90,2] + 112.425;
   1:L PR[91] 10mm/sec FINE;
   1:  PR[GP1:91,1] = PR[GP1:90,1] + 97.732;
   1:  PR[GP1:91,2] = PR[GP1:90,2] + 111.605;
   1:L PR[91] 10mm/sec FINE;
   1:  PR[GP1:91,1] = PR[GP1:90,1] + 96.773;
   1:  PR[GP1:91,2] = PR[GP1:90,2] + 110.811;
   1:L PR[91] 10mm/sec FINE;
   1:  PR[GP1:91,1] = PR[GP1:90,1] + 95.610;
   1:  PR[GP1:91,2] = PR[GP1:90,2] + 110.537;
   1:L PR[91] 10mm/sec FINE;
   1:  PR[GP1:91,1] = PR[GP1:90,1] + 95.213;
   1:  PR[GP1:91,2] = PR[GP1:90,2] + 110.532;
   1:L PR[91] 10mm/sec FINE;
   1:  PR[GP1:91,1] = PR[GP1:90,1] + 94.846;
   1:  PR[GP1:91,2] = PR[GP1:90,2] + 110.622;
   1:L PR[91] 10mm/sec FINE;
   1:  PR[GP1:91,1] = PR[GP1:90,1] + 94.513;
   1:  PR[GP1:91,2] = PR[GP1:90,2] + 110.667;
   1:L PR[91] 10mm/sec FINE;
   1:  PR[GP1:91,1] = PR[GP1:90,1] + 94.262;
   1:  PR[GP1:91,2] = PR[GP1:90,2] + 110.734;
   1:L PR[91] 10mm/sec FINE;
   1:  PR[GP1:91,1] = PR[GP1:90,1] + 94.003;
   1:  PR[GP1:91,2] = PR[GP1:90,2] + 110.850;
   1:L PR[91] 10mm/sec FINE;
   1:  PR[GP1:91,1] = PR[GP1:90,1] + 93.356;
   1:  PR[GP1:91,2] = PR[GP1:90,2] + 111.376;
   1:L PR[91] 10mm/sec FINE;
   1:  PR[GP1:91,1] = PR[GP1:90,1] + 93.209;
   1:  PR[GP1:91,2] = PR[GP1:90,2] + 111.514;
   1:L PR[91] 10mm/sec FINE;
   1:  PR[GP1:91,1] = PR[GP1:90,1] + 93.095;
   1:  PR[GP1:91,2] = PR[GP1:90,2] + 111.660;
   1:L PR[91] 10mm/sec FINE;
   1:  PR[GP1:91,1] = PR[GP1:90,1] + 92.794;
   1:  PR[GP1:91,2] = PR[GP1:90,2] + 112.356;
   1:L PR[91] 10mm/sec FINE;
   1:  PR[GP1:91,1] = PR[GP1:90,1] + 92.723;
   1:  PR[GP1:91,2] = PR[GP1:90,2] + 112.487;
   1:L PR[91] 10mm/sec FINE;
   1:  PR[GP1:91,1] = PR[GP1:90,1] + 92.689;
   1:  PR[GP1:91,2] = PR[GP1:90,2] + 112.597;
   1:L PR[91] 10mm/sec FINE;
   1:  PR[GP1:91,1] = PR[GP1:90,1] + 92.630;
   1:  PR[GP1:91,2] = PR[GP1:90,2] + 112.600;
   1:L PR[91] 10mm/sec FINE;
   1:  PR[GP1:91,1] = PR[GP1:90,1] + 92.333;
   1:  PR[GP1:91,2] = PR[GP1:90,2] + 113.722;
   1:L PR[91] 10mm/sec FINE;
   1:  PR[GP1:91,1] = PR[GP1:90,1] + 92.194;
   1:  PR[GP1:91,2] = PR[GP1:90,2] + 114.354;
   1:L PR[91] 10mm/sec FINE;
   1:  PR[GP1:91,1] = PR[GP1:90,1] + 91.774;
   1:  PR[GP1:91,2] = PR[GP1:90,2] + 115.804;
   1:L PR[91] 10mm/sec FINE;
   1:  PR[GP1:91,1] = PR[GP1:90,1] + 91.062;
   1:  PR[GP1:91,2] = PR[GP1:90,2] + 117.384;
   1:L PR[91] 10mm/sec FINE;
   1:  PR[GP1:91,1] = PR[GP1:90,1] + 90.410;
   1:  PR[GP1:91,2] = PR[GP1:90,2] + 118.595;
   1:L PR[91] 10mm/sec FINE;
   1:  PR[GP1:91,1] = PR[GP1:90,1] + 89.397;
   1:  PR[GP1:91,2] = PR[GP1:90,2] + 120.114;
   1:L PR[91] 10mm/sec FINE;
   1:  PR[GP1:91,1] = PR[GP1:90,1] + 88.598;
   1:  PR[GP1:91,2] = PR[GP1:90,2] + 121.050;
   1:L PR[91] 10mm/sec FINE;
   1:  PR[GP1:91,1] = PR[GP1:90,1] + 87.288;
   1:  PR[GP1:91,2] = PR[GP1:90,2] + 122.450;
   1:L PR[91] 10mm/sec FINE;
   1:  PR[GP1:91,1] = PR[GP1:90,1] + 84.824;
   1:  PR[GP1:91,2] = PR[GP1:90,2] + 124.334;
   1:L PR[91] 10mm/sec FINE;
   1:  PR[GP1:91,1] = PR[GP1:90,1] + 83.056;
   1:  PR[GP1:91,2] = PR[GP1:90,2] + 125.274;
   1:L PR[91] 10mm/sec FINE;
   1:  PR[GP1:91,1] = PR[GP1:90,1] + 82.106;
   1:  PR[GP1:91,2] = PR[GP1:90,2] + 125.723;
   1:L PR[91] 10mm/sec FINE;
   1:  PR[GP1:91,1] = PR[GP1:90,1] + 80.138;
   1:  PR[GP1:91,2] = PR[GP1:90,2] + 126.384;
   1:L PR[91] 10mm/sec FINE;
   1:  PR[GP1:91,1] = PR[GP1:90,1] + 79.220;
   1:  PR[GP1:91,2] = PR[GP1:90,2] + 126.598;
   1:L PR[91] 10mm/sec FINE;
   1:  PR[GP1:91,1] = PR[GP1:90,1] + 77.110;
   1:  PR[GP1:91,2] = PR[GP1:90,2] + 126.937;
   1:L PR[91] 10mm/sec FINE;
   1:  PR[GP1:91,1] = PR[GP1:90,1] + 74.965;
   1:  PR[GP1:91,2] = PR[GP1:90,2] + 126.925;
   1:L PR[91] 10mm/sec FINE;
   1:  PR[GP1:91,1] = PR[GP1:90,1] + 74.057;
   1:  PR[GP1:91,2] = PR[GP1:90,2] + 126.940;
   1:L PR[91] 10mm/sec FINE;
   1:  PR[GP1:91,1] = PR[GP1:90,1] + 71.898;
   1:  PR[GP1:91,2] = PR[GP1:90,2] + 126.568;
   1:L PR[91] 10mm/sec FINE;
   1:  PR[GP1:91,1] = PR[GP1:90,1] + 71.084;
   1:  PR[GP1:91,2] = PR[GP1:90,2] + 126.408;
   1:L PR[91] 10mm/sec FINE;
   1:  PR[GP1:91,1] = PR[GP1:90,1] + 68.977;
   1:  PR[GP1:91,2] = PR[GP1:90,2] + 125.674;
   1:L PR[91] 10mm/sec FINE;
   1:  PR[GP1:91,1] = PR[GP1:90,1] + 68.269;
   1:  PR[GP1:91,2] = PR[GP1:90,2] + 125.370;
   1:L PR[91] 10mm/sec FINE;
   1:  PR[GP1:91,1] = PR[GP1:90,1] + 66.283;
   1:  PR[GP1:91,2] = PR[GP1:90,2] + 124.285;
   1:L PR[91] 10mm/sec FINE;
   1:  PR[GP1:91,1] = PR[GP1:90,1] + 65.689;
   1:  PR[GP1:91,2] = PR[GP1:90,2] + 123.863;
   1:L PR[91] 10mm/sec FINE;
   1:  PR[GP1:91,1] = PR[GP1:90,1] + 63.889;
   1:  PR[GP1:91,2] = PR[GP1:90,2] + 122.454;
   1:L PR[91] 10mm/sec FINE;
   1:  PR[GP1:91,1] = PR[GP1:90,1] + 61.859;
   1:  PR[GP1:91,2] = PR[GP1:90,2] + 120.235;
   1:L PR[91] 10mm/sec FINE;
   1:  PR[GP1:91,1] = PR[GP1:90,1] + 60.604;
   1:  PR[GP1:91,2] = PR[GP1:90,2] + 118.306;
   1:L PR[91] 10mm/sec FINE;
   1:  PR[GP1:91,1] = PR[GP1:90,1] + 60.252;
   1:  PR[GP1:91,2] = PR[GP1:90,2] + 117.705;
   1:L PR[91] 10mm/sec FINE;
   1:  PR[GP1:91,1] = PR[GP1:90,1] + 59.328;
   1:  PR[GP1:91,2] = PR[GP1:90,2] + 115.589;
   1:L PR[91] 10mm/sec FINE;
   1:  PR[GP1:91,1] = PR[GP1:90,1] + 59.112;
   1:  PR[GP1:91,2] = PR[GP1:90,2] + 114.934;
   1:L PR[91] 10mm/sec FINE;
   1:  PR[GP1:91,1] = PR[GP1:90,1] + 58.548;
   1:  PR[GP1:91,2] = PR[GP1:90,2] + 112.698;
   1:L PR[91] 10mm/sec FINE;
   1:  PR[GP1:91,1] = PR[GP1:90,1] + 58.357;
   1:  PR[GP1:91,2] = PR[GP1:90,2] + 110.389;
   1:L PR[91] 10mm/sec FINE;
   1:  PR[GP1:91,1] = PR[GP1:90,1] + 58.285;
   1:  PR[GP1:91,2] = PR[GP1:90,2] + 109.704;
   1:L PR[91] 10mm/sec FINE;
   1:  PR[GP1:91,1] = PR[GP1:90,1] + 58.474;
   1:  PR[GP1:91,2] = PR[GP1:90,2] + 107.410;
   1:L PR[91] 10mm/sec FINE;
   1:  PR[GP1:91,1] = PR[GP1:90,1] + 58.550;
   1:  PR[GP1:91,2] = PR[GP1:90,2] + 106.710;
   1:L PR[91] 10mm/sec FINE;
   1:  PR[GP1:91,1] = PR[GP1:90,1] + 59.110;
   1:  PR[GP1:91,2] = PR[GP1:90,2] + 104.491;
   1:L PR[91] 10mm/sec FINE;
   1:  PR[GP1:91,1] = PR[GP1:90,1] + 59.338;
   1:  PR[GP1:91,2] = PR[GP1:90,2] + 103.798;
   1:L PR[91] 10mm/sec FINE;
   1:  PR[GP1:91,1] = PR[GP1:90,1] + 60.245;
   1:  PR[GP1:91,2] = PR[GP1:90,2] + 101.721;
   1:L PR[91] 10mm/sec FINE;
   1:  PR[GP1:91,1] = PR[GP1:90,1] + 60.636;
   1:  PR[GP1:91,2] = PR[GP1:90,2] + 101.056;
   1:L PR[91] 10mm/sec FINE;
   1:  PR[GP1:91,1] = PR[GP1:90,1] + 61.856;
   1:  PR[GP1:91,2] = PR[GP1:90,2] + 99.182;
   1:L PR[91] 10mm/sec FINE;
   1:  PR[GP1:91,1] = PR[GP1:90,1] + 63.904;
   1:  PR[GP1:91,2] = PR[GP1:90,2] + 96.947;
   1:L PR[91] 10mm/sec FINE;
   1:  PR[GP1:91,1] = PR[GP1:90,1] + 65.632;
   1:  PR[GP1:91,2] = PR[GP1:90,2] + 95.592;
   1:L PR[91] 10mm/sec FINE;
   1:  PR[GP1:91,1] = PR[GP1:90,1] + 66.333;
   1:  PR[GP1:91,2] = PR[GP1:90,2] + 95.097;
   1:L PR[91] 10mm/sec FINE;
   1:  PR[GP1:91,1] = PR[GP1:90,1] + 68.017;
   1:  PR[GP1:91,2] = PR[GP1:90,2] + 94.178;
   1:  PR[GP1:91,3] = PR[GP1:90,3] + 6.900;
   1:L PR[91] 10mm/sec FINE;
   1:  PR[GP1:91,1] = PR[GP1:90,1] + 69.517;
   1:  PR[GP1:91,2] = PR[GP1:90,2] + 93.539;
   1:L PR[91] 10mm/sec FINE;
   1:  PR[GP1:91,1] = PR[GP1:90,1] + 70.963;
   1:  PR[GP1:91,2] = PR[GP1:90,2] + 93.036;
   1:L PR[91] 10mm/sec FINE;
   1:  PR[GP1:91,1] = PR[GP1:90,1] + 72.481;
   1:  PR[GP1:91,2] = PR[GP1:90,2] + 92.775;
   1:L PR[91] 10mm/sec FINE;
   1:  PR[GP1:91,1] = PR[GP1:90,1] + 74.140;
   1:  PR[GP1:91,2] = PR[GP1:90,2] + 92.451;
   1:L PR[91] 10mm/sec FINE;
   1:  PR[GP1:91,1] = PR[GP1:90,1] + 75.548;
   1:  PR[GP1:91,2] = PR[GP1:90,2] + 92.443;
   1:L PR[91] 10mm/sec FINE;
   1:  PR[GP1:91,1] = PR[GP1:90,1] + 77.440;
   1:  PR[GP1:91,2] = PR[GP1:90,2] + 92.483;
   1:L PR[91] 10mm/sec FINE;
   1:  PR[GP1:91,1] = PR[GP1:90,1] + 78.689;
   1:  PR[GP1:91,2] = PR[GP1:90,2] + 92.684;
   1:L PR[91] 10mm/sec FINE;
   1:  PR[GP1:91,1] = PR[GP1:90,1] + 80.757;
   1:  PR[GP1:91,2] = PR[GP1:90,2] + 93.176;
   1:L PR[91] 10mm/sec FINE;
   1:  PR[GP1:91,1] = PR[GP1:90,1] + 81.808;
   1:  PR[GP1:91,2] = PR[GP1:90,2] + 93.529;
   1:L PR[91] 10mm/sec FINE;
   1:  PR[GP1:91,1] = PR[GP1:90,1] + 83.951;
   1:  PR[GP1:91,2] = PR[GP1:90,2] + 94.552;
   1:L PR[91] 10mm/sec FINE;
   1:  PR[GP1:91,1] = PR[GP1:90,1] + 84.789;
   1:  PR[GP1:91,2] = PR[GP1:90,2] + 94.998;
   1:L PR[91] 10mm/sec FINE;
   1:  PR[GP1:91,1] = PR[GP1:90,1] + 87.499;
   1:  PR[GP1:91,2] = PR[GP1:90,2] + 97.081;
   1:L PR[91] 10mm/sec FINE;
   1:  PR[GP1:91,1] = PR[GP1:90,1] + 88.047;
   1:  PR[GP1:91,2] = PR[GP1:90,2] + 97.666;
   1:L PR[91] 10mm/sec FINE;
   1:  PR[GP1:91,1] = PR[GP1:90,1] + 89.777;
   1:  PR[GP1:91,2] = PR[GP1:90,2] + 99.714;
   1:L PR[91] 10mm/sec FINE;
   1:  PR[GP1:91,1] = PR[GP1:90,1] + 90.159;
   1:  PR[GP1:91,2] = PR[GP1:90,2] + 100.287;
   1:L PR[91] 10mm/sec FINE;
   1:  PR[GP1:91,1] = PR[GP1:90,1] + 91.486;
   1:  PR[GP1:91,2] = PR[GP1:90,2] + 102.774;
   1:L PR[91] 10mm/sec FINE;
   1:  PR[GP1:91,1] = PR[GP1:90,1] + 91.744;
   1:  PR[GP1:91,2] = PR[GP1:90,2] + 103.346;
   1:L PR[91] 10mm/sec FINE;
   1:  PR[GP1:91,1] = PR[GP1:90,1] + 92.345;
   1:  PR[GP1:91,2] = PR[GP1:90,2] + 105.594;
   1:L PR[91] 10mm/sec FINE;
   1:  PR[GP1:91,1] = PR[GP1:90,1] + 92.697;
   1:  PR[GP1:91,2] = PR[GP1:90,2] + 106.808;
   1:L PR[91] 10mm/sec FINE;
   1:  PR[GP1:91,1] = PR[GP1:90,1] + 92.800;
   1:  PR[GP1:91,2] = PR[GP1:90,2] + 106.950;
   1:L PR[91] 10mm/sec FINE;
   1:  PR[GP1:91,1] = PR[GP1:90,1] + 93.034;
   1:  PR[GP1:91,2] = PR[GP1:90,2] + 107.524;
   1:L PR[91] 10mm/sec FINE;
   1:  PR[GP1:91,1] = PR[GP1:90,1] + 93.153;
   1:  PR[GP1:91,2] = PR[GP1:90,2] + 107.753;
   1:L PR[91] 10mm/sec FINE;
   1:  PR[GP1:91,1] = PR[GP1:90,1] + 93.343;
   1:  PR[GP1:91,2] = PR[GP1:90,2] + 108.009;
